// TwinCAT 3 PLC project Untitled1
// ProgramVersion: 3.1.4023.0
// libraries:
//   Tc2_MC2, * (Beckhoff Automation GmbH)
//   Tc2_Standard, * (Beckhoff Automation GmbH)
//   Tc2_System, * (Beckhoff Automation GmbH)
//   Tc2_Utilities, * (Beckhoff Automation GmbH)
//   Tc3_JsonXml, * (Beckhoff Automation GmbH)
//   Tc3_Module, * (Beckhoff Automation GmbH)
// project tree:
//   DUTs/ Bundle.TcDUT, Interval.TcDUT (not stored), PositionMaterials.TcDUT, SuctionPad.TcDUT
//   DUTs/Enums/ A22.TcDUT (not stored), Cardboard.TcDUT (not stored), CornerGuard.TcDUT (not stored), Homing.TcDUT (not stored), SectionEnum.TcDUT, Surface.TcDUT
//   DUTs/Insertion/ABSTRACT/ FBA_Drive.TcPOU, I_ContinuousDrive.TcIO (not stored), I_Drive.TcIO, I_EncodedDrive.TcIO (not stored), I_PositionalDrive.TcIO (not stored)
//   DUTs/Insertion/Drives/ ClearLinkMC.TcPOU, ServoNC.TcPOU, SimplePiston.TcPOU (not stored)
//   DUTs/Insertion/ Insertion.TcPOU
//   DUTs/Machines/ FoldingMachine.TcPOU, KukaRobot.TcPOU (not stored), RobotA22.TcPOU (not stored), WrapMachine.TcPOU (not stored)
//   DUTs/Material Holders/ MaterialHolder.TcPOU (not stored), MaterialSlot.TcDUT, SkidMagazine.TcPOU (not stored)
//   GVLs/ ContainerArrays.TcGVL, GVL.TcGVL (not stored), Hardware.TcGVL, Misc.TcGVL (not stored)
//   / PlcTask.TcTTO
//   POUs/A22 - Cardboard-Corner Guard/AOIs/ AOI_LoadCornerCardboard.TcPOU, AOI_LoadCornerGuard.TcPOU, AOI_LoadFlatCardboard.TcPOU
//   POUs/A22 - Cardboard-Corner Guard/ FiberboardEx.TcPOU
//   POUs/ FB_System.TcPOU, MAIN.TcPOU, BundleToJson.TcPOU
//   POUs/Hardware Calls/ SuctionQualityPtrArr.TcPOU (not stored), SetSuctionsPtrArr.TcPOU (not stored), CallHardwareModules.TcPOU, SuctionQuality.TcPOU (not stored), SetSuctions.TcPOU, SetupHardware.TcPOU (not stored)
//   POUs/Materials/ GetMaterialLength.TcPOU, GetMaterialLengthFromCode.TcPOU (not stored), GetPairMasterLength.TcPOU (not stored), GetPositionMasterLength.TcPOU (not stored), MatchesMaterialType.TcPOU
//   POUs/Utility/ CEILING.TcPOU (not stored), IntegerBitAccess.TcPOU (not stored), IntegerToBoolArray.TcPOU (not stored), WithinTolerance.TcPOU (not stored)
// real-time tasks:
//   TASK PlcTask: cycle T#10ms, priority 20, ADS port 350
// motion (NC):
//   TASK NC-Task 1 SAF: cycle T#2ms, priority 4, ADS port 501
//   TASK NC-Task 1 SVB: cycle T#10ms, priority 8, ADS port 511
//   AXIS A22_IM_HS_L (id 1)
//     OtherSettings: AllowMotionCmdToSlave=true
//     encoder EncType=1
//     drive DrvType=5
//       Analog: TorqueSetpointScale=10, ScaleFactorActTorque=0.1
//       TimeComp: TaskDelayCycles=1
//     controller CtrType=1
//       CtrPara: PriorControlFactor=1
//         Observer: BandWidth=20
//   AXIS A22_IM_HS_R (id 2)
//     OtherSettings: AllowMotionCmdToSlave=true
//     encoder EncType=19
//       EncPara: MaxCount=#xffffffff
//     drive DrvType=16
//       DrvPara: MaxCount=#xffffffff, DriveControlDWord=#x00000100
//         Analog: TorqueSetpointScale=10, ScaleFactorActTorque=0.1
//         TimeComp: TaskDelayCycles=1
//     controller CtrType=1
//       CtrPara: PriorControlFactor=1
//         Observer: BandWidth=20
// I/O:
//   DEVICE Device 2 (TC3 EIP Scanner), AmsNetId 5.131.216.41.4.1
//     ClearLink_A22 // <INFO> 169.254.0.152, ClearLink (ProdCode: 1, Rev: 2.93, Mac: 24:15:10:b0:30:37) </INFO> <EDS> C:\TwinCAT\3.1\Config\Io\EtherNetIP\clearlink_2.92.eds </EDS>
//   DEVICE Device 1 (EtherCAT), AmsNetId 5.131.216.41.2.1
//     EK1200 [EK1200-5000 EtherCAT Power supply (2A E-Bus)]
//       IPC_O [EL2809 16Ch. Dig. Output 24V, 0.5A]
//       JUNC_1 [EK1122 2 port EtherCAT junction]
//         A21_C4 [EK1100 EtherCAT Coupler (2A E-Bus)]
//           A21_C4_I1 [EL1809 16Ch. Dig. Input 24V, 3ms]
//           A21_C4_O2 [EL2809 16Ch. Dig. Output 24V, 0.5A]
//           A21_C4_O3 [EL2809 16Ch. Dig. Output 24V, 0.5A]
//           BRIDGE_ROBOT1 [EL6695 EtherCAT Bridge terminal (Primary)]
//           A21_C4_END [EL9011 End Terminal]
//         A21_SB01 [EP1809-0021 16 Ch. Dig. Input 24V, 3ms, M8]
//         A21_SB05 [EP1008-0001 8 Ch. Dig. Input 24V, 3ms, M8]
//         A21_SB04 [EP1809-0021 16 Ch. Dig. Input 24V, 3ms, M8]
//         A21_SB03 [EP1008-0001 8 Ch. Dig. Input 24V, 3ms, M8]
//         A21_C1 [EK1100 EtherCAT Coupler (2A E-Bus)]
//           A21_C1_I1 [EL1809 16Ch. Dig. Input 24V, 3ms]
//           A21_C1_O2 [EL2809 16Ch. Dig. Output 24V, 0.5A]
//           BRIDGE_ROBOT2 [EL6695 EtherCAT Bridge terminal (Primary)]
//           A21_C1_END [EL9011 End Terminal]
//         A21_SB02 [EP1809-0021 16 Ch. Dig. Input 24V, 3ms, M8]
//         A21_SB07 [EP1008-0001 8 Ch. Dig. Input 24V, 3ms, M8]
//         A21_SB06 [EP1008-0001 8 Ch. Dig. Input 24V, 3ms, M8]
//       JUNC_2 [EK1122 2 port EtherCAT junction]
//         A22_C1 [EK1100 EtherCAT Coupler (2A E-Bus)]
//           A22_C1_I1 [EL1809 16Ch. Dig. Input 24V, 3ms]
//           A22_C1_O2 [EL2809 16Ch. Dig. Output 24V, 0.5A]
//           A22_C1_JUNC [EK1122 2 port EtherCAT junction]
//             A22_C4 [EK1100 EtherCAT Coupler (2A E-Bus)]
//               A22_C4_I1 [EL1809 16Ch. Dig. Input 24V, 3ms]
//               A22_C4_O2 [EL2809 16Ch. Dig. Output 24V, 0.5A]
//               A22_C4_O3 [EL2809 16Ch. Dig. Output 24V, 0.5A]
//               Term 31 (EL9011) [EL9011 End Terminal]
//             A22_C4_NC2 [CD02 EtherCAT Drive (CoE)]
//             A22_C4_NC1_TEMP [EK1100 EtherCAT Coupler (2A E-Bus)]
//               Term 34 (EL1008) [EL1008 8Ch. Dig. Input 24V, 3ms]
//               Term 35 (EL2008) [EL2008 8Ch. Dig. Output 24V, 0.5A]
//               Term 36 (EL9011) [EL9011 End Terminal]
//             A22_SB01 [EP1809-0021 16 Ch. Dig. Input 24V, 3ms, M8]
//             A22_SB04 [EP1809-0021 16 Ch. Dig. Input 24V, 3ms, M8]
//             A22_SB05 [EP1008-0001 8 Ch. Dig. Input 24V, 3ms, M8]
//             A22_C5 [EK1100 EtherCAT Coupler (2A E-Bus)]
//               A22_C5_I1 [EL1809 16Ch. Dig. Input 24V, 3ms]
//               A22_C5_O2 [EL2809 16Ch. Dig. Output 24V, 0.5A]
//               A22_C5_END [EL9011 End Terminal]
//             A22_SB06 [EP1008-0001 8 Ch. Dig. Input 24V, 3ms, M8]
//             A22_C6 [EK1100 EtherCAT Coupler (2A E-Bus)]
//               A22_C6_I1 [EL1809 16Ch. Dig. Input 24V, 3ms]
//               A22_C6_O2 [EL2809 16Ch. Dig. Output 24V, 0.5A]
//               A22_C6_O3 [EL2809 16Ch. Dig. Output 24V, 0.5A]
//               BRDIGE_ROBOT3 [EL6695 EtherCAT Bridge terminal (Primary)]
//               A22_C6_END [EL9011 End Terminal]
//             A22_SB08 [EP1008-0001 8 Ch. Dig. Input 24V, 3ms, M8]
//             A22_SB09 [EP2338-1001 8 Ch. Dig. Input/Output 24V, 3ms, 0,5A, M8]
//             A22_SB03 [EP1008-0001 8 Ch. Dig. Input 24V, 3ms, M8]
//             A22_SB02 [EP1809-0021 16 Ch. Dig. Input 24V, 3ms, M8]
//             A22_SB07 [EP1008-0001 8 Ch. Dig. Input 24V, 3ms, M8]
//             A22_C7 [EK1100 EtherCAT Coupler (2A E-Bus)]
//               A22_C7_I1 [EL1809 16Ch. Dig. Input 24V, 3ms]
//               A22_C7_O2 [EL2809 16Ch. Dig. Output 24V, 0.5A]
//               BRIDGE_ROBOT4 [EL6695 EtherCAT Bridge terminal (Primary)]
//               A22_C7_END [EL9011 End Terminal]
// variable links:
//   NC-Task 1 SAF/Axes/A22_IM_HS_R <-> Device 1 (EtherCAT)/EK1200/JUNC_2/A22_C1/A22_C1_JUNC/A22_C4_NC2
//     Drive/Inputs/In/nDataIn1 <-> TxPDO 1/Following Error Actual Value
//     Drive/Inputs/In/nDataIn3[0] <-> TxPDO 4/Torque Actual Value
//     Drive/Inputs/In/nDcOutputTime <-> InfoData/DcOutputShift
//     Drive/Inputs/In/nState1 <-> TxPDO 4/Statusword
//     Drive/Inputs/In/nState2 <-> TxPDO 4/Statusword @bit 8
//     Drive/Inputs/In/nState4 @bit 1 <-> WcState/InputToggle
//     Drive/Inputs/In/nState4 <-> WcState/WcState
//     Drive/Inputs/In/nState5 <-> TxPDO 3/Modes of Operation Display
//     Drive/Outputs/Out/nCtrl1 <-> RxPDO 4/Controlword
//     Drive/Outputs/Out/nCtrl2 <-> RxPDO 4/Controlword @bit 8
//     Drive/Outputs/Out/nCtrl5 <-> RxPDO 4/Modes of Operation
//     Drive/Outputs/Out/nDataOut1 <-> RxPDO 1/Target Position
//     Drive/Outputs/Out/nDataOut2 <-> RxPDO 2/Target Velocity
//     Drive/Outputs/Out/nDataOut3[0] <-> RxPDO 4/Torque Offset
//     Drive/Outputs/Out/nDataOut4[0] <-> RxPDO 3/Target Torque
//     Enc/Inputs/In/nDataIn1 <-> TxPDO 2/Position Actual Value
//     Enc/Inputs/In/nDcInputTime <-> InfoData/DcInputShift
//     Enc/Inputs/In/nState4 @bit 1 <-> WcState/InputToggle
//     Enc/Inputs/In/nState4 <-> WcState/WcState
//   Untitled1/Untitled1 Instance <-> Device 1 (EtherCAT)/EK1200/JUNC_2/A22_C1/A22_C1_JUNC/A22_C4/A22_C4_O3
//     PlcTask Outputs/Hardware.verticalDriveA22Right.brakeRelease <-> Channel 1/Output
//   Untitled1/Untitled1 Instance <-> Device 1 (EtherCAT)/EK1200/JUNC_2/A22_C1/A22_C1_JUNC/A22_C6/BRDIGE_ROBOT3
//     PlcTask Inputs/Hardware.robot3.inputs[{2..20}] <-> IO Inputs/In_{2..20}  (19 links)
//     PlcTask Inputs/Hardware.robot3.inputs[1] <-> IO Inputs/In
//     PlcTask Inputs/Hardware.robot3.offline <-> SYNC Inputs/External device not connected
//     PlcTask Outputs/Hardware.robot3.outputs[{2..20}] <-> IO Outputs/Out_{2..20}  (19 links)
//     PlcTask Outputs/Hardware.robot3.outputs[1] <-> IO Outputs/Out
//   Untitled1/Untitled1 Instance <-> Device 1 (EtherCAT)/EK1200/JUNC_2/A22_C1/A22_C1_JUNC/A22_C7/BRIDGE_ROBOT4
//     PlcTask Inputs/Hardware.robot4.inputs[{2..20}] <-> IO Inputs/In_{2..20}  (19 links)
//     PlcTask Inputs/Hardware.robot4.inputs[1] <-> IO Inputs/In
//     PlcTask Inputs/Hardware.robot4.offline <-> SYNC Inputs/External device not connected
//     PlcTask Outputs/Hardware.robot4.outputs[{2..20}] <-> IO Outputs/Out_{2..20}  (19 links)
//     PlcTask Outputs/Hardware.robot4.outputs[1] <-> IO Outputs/Out
//   Untitled1/Untitled1 Instance <-> Device 1 (EtherCAT)/EK1200/JUNC_2/A22_C1/A22_C1_JUNC/A22_SB01
//     PlcTask Inputs/Hardware.horizontalDriveA22Left.home <-> Channel 6/Input
//     PlcTask Inputs/Hardware.horizontalDriveA22Left.innerLimit <-> Channel 5/Input
//     PlcTask Inputs/Hardware.horizontalDriveA22Left.outerLimit <-> Channel 4/Input
//     PlcTask Inputs/Hardware.suctionA22BottomLeft[1].occupied <-> Channel 10/Input
//     PlcTask Inputs/Hardware.suctionA22BottomLeft[2].occupied <-> Channel 11/Input
//     PlcTask Inputs/Hardware.suctionA22BottomLeft[3].occupied <-> Channel 12/Input
//     PlcTask Inputs/Hardware.suctionA22TopLeft[1].occupied <-> Channel 7/Input
//     PlcTask Inputs/Hardware.suctionA22TopLeft[2].occupied <-> Channel 8/Input
//     PlcTask Inputs/Hardware.suctionA22TopLeft[3].occupied <-> Channel 9/Input
//     PlcTask Inputs/Hardware.verticalDriveA22Left.home <-> Channel 3/Input
//     PlcTask Inputs/Hardware.verticalDriveA22Left.innerLimit <-> Channel 2/Input
//     PlcTask Inputs/Hardware.verticalDriveA22Left.outerLimit <-> Channel 1/Input
//   Untitled1/Untitled1 Instance <-> Device 1 (EtherCAT)/EK1200/JUNC_2/A22_C1/A22_C1_JUNC/A22_SB02
//     PlcTask Inputs/Hardware.horizontalDriveA22Right.home <-> Channel 6/Input
//     PlcTask Inputs/Hardware.horizontalDriveA22Right.innerLimit <-> Channel 4/Input
//     PlcTask Inputs/Hardware.horizontalDriveA22Right.outerLimit <-> Channel 5/Input
//     PlcTask Inputs/Hardware.suctionA22BottomRight[1].occupied <-> Channel 10/Input
//     PlcTask Inputs/Hardware.suctionA22BottomRight[2].occupied <-> Channel 11/Input
//     PlcTask Inputs/Hardware.suctionA22BottomRight[3].occupied <-> Channel 12/Input
//     PlcTask Inputs/Hardware.suctionA22TopRight[1].occupied <-> Channel 7/Input
//     PlcTask Inputs/Hardware.suctionA22TopRight[2].occupied <-> Channel 8/Input
//     PlcTask Inputs/Hardware.suctionA22TopRight[3].occupied <-> Channel 9/Input
//     PlcTask Inputs/Hardware.verticalDriveA22Right.home <-> Channel 3/Input
//     PlcTask Inputs/Hardware.verticalDriveA22Right.innerLimit <-> Channel 2/Input
//     PlcTask Inputs/Hardware.verticalDriveA22Right.outerLimit <-> Channel 1/Input
//   Untitled1/Untitled1 Instance <-> Device 1 (EtherCAT)/EK1200/JUNC_2/A22_C1/A22_C1_JUNC/A22_SB06
//     PlcTask Inputs/Hardware.magazineA22Left.inPosition[1] <-> Channel 7/Input
//     PlcTask Inputs/Hardware.magazineA22Left.inPosition[2] <-> Channel 8/Input
//   Untitled1/Untitled1 Instance <-> Device 2 (TC3 EIP Scanner)/ClearLink_A22
//     PlcTask Inputs/Hardware.verticalDriveA22Left.hlfb <-> Connection 1 (Input/Output)/Inputs/Motor0 HLFB Duty
//     PlcTask Inputs/Hardware.verticalDriveA22Right.hlfb <-> Connection 1 (Input/Output)/Inputs/Motor1 HLFB Duty
//     PlcTask Outputs/Hardware.verticalDriveA22Left.outputRegister <-> Connection 1 (Input/Output)/Outputs/Motor0 Out Reg
//     PlcTask Outputs/Hardware.verticalDriveA22Left.pulse <-> Connection 1 (Input/Output)/Outputs/Motor0 Trig Pulses
//     PlcTask Outputs/Hardware.verticalDriveA22Right.outputRegister <-> Connection 1 (Input/Output)/Outputs/Motor1 Out Reg
//     PlcTask Outputs/Hardware.verticalDriveA22Right.pulse <-> Connection 1 (Input/Output)/Outputs/Motor1 Trig Pulses
//   Untitled1/Untitled1 Instance <-> NC-Task 1 SAF/Axes/A22_IM_HS_L
//     PlcTask Inputs/Hardware.horizontalDriveA22Left.axis.NcToPlc <-> Outputs/ToPlc
//     PlcTask Outputs/Hardware.horizontalDriveA22Left.axis.PlcToNc <-> Inputs/FromPlc
//   Untitled1/Untitled1 Instance <-> NC-Task 1 SAF/Axes/A22_IM_HS_R
//     PlcTask Inputs/Hardware.horizontalDriveA22Right.axis.NcToPlc <-> Outputs/ToPlc
//     PlcTask Outputs/Hardware.horizontalDriveA22Right.axis.PlcToNc <-> Inputs/FromPlc

CONFIGURATION Untitled1
    RESOURCE PLC ON TwinCAT3
        TASK PlcTask(INTERVAL := T#10ms, PRIORITY := 20);
        PROGRAM MAIN WITH PlcTask : MAIN;
    END_RESOURCE
END_CONFIGURATION

// ---- DUTs/Bundle.TcDUT
{attribute 'enable_dynamic_creation'}
TYPE Bundle :
STRUCT
	id : STRING;
	weight : REAL;
	
	length : INT;
	width : INT;
	height : INT;
	
	pieces : INT;
	layers : INT;
	piecesPerLayer : INT;
	
	extrusionWeight : INT;
	extrusionHeight : INT;
	extrusionWidth : INT;
	
	//if a process is true, send it to the correct area and turn it false when complete
	reqProcesses : ARRAY[0..3] OF BOOL; //this may not be used
	
	manRE, autoRE : BOOL; //repacking - coming soon
	manSS, autoSS : BOOL; //packaging
	
	paperFront : BOOL;
	paperBack : BOOL;
	cardboardFront : BOOL;
	cardboardBack : BOOL;
	
	paperTop : ARRAY[0..GVL.maxPairs] OF Interval;
	paperLeft : ARRAY[0..GVL.maxPairs] OF Interval;
	paperRight : ARRAY[0..GVL.maxPairs] OF Interval;
	paperBottom : ARRAY[0..GVL.maxPairs] OF Interval;
		
	cardboard : ARRAY[0..GVL.maxPairs] OF PositionMaterials;
	cardboardTopLeftFold : ARRAY[0..GVL.maxPairs] OF INT;
	cardboardTopRightFold : ARRAY[0..GVL.maxPairs] OF INT;
	cardboardBottomLeftFold : ARRAY[0..GVL.maxPairs] OF INT;
	cardboardBottomRightFold : ARRAY[0..GVL.maxPairs] OF INT;
	
	topLeftFolds : ARRAY[0..GVL.maxPairs] OF INT;
	topRightFolds : ARRAY[0..GVL.maxPairs] OF INT;
	bottomLeftFolds : ARRAY[0..GVL.maxPairs] OF INT;
	bottomRightFolds : ARRAY[0..GVL.maxPairs] OF INT;
	
	cornerGuard : ARRAY[0..GVL.maxPairs] OF PositionMaterials;
	
	chipboard : ARRAY[0..GVL.maxPairs] OF PositionMaterials;
	woodBunk : ARRAY[0..GVL.maxPairs] OF PositionMaterials;
	
	cardboard_over_cornerGuard : BOOL;
	
	currStep : USINT; //for runtime use only
	
	//for production log database
	
	timeStart : TIMESTRUCT;
	timeDone : TIMESTRUCT;
END_STRUCT
END_TYPE

// ---- DUTs/Enums/SectionEnum.TcDUT
{attribute 'qualified_only'}
TYPE SectionEnum :
(
	NULL_SECTION := 0,
	PAPER,
	CARDBOARD_CORNERGUARD,
	CHIPBOARD,
	WOOD_BUNK,
	OUTPUT,
	
	size
);
END_TYPE

// ---- DUTs/Enums/Surface.TcDUT
{attribute 'qualified_only'}
//{attribute 'strict'}
TYPE Surface :
(
	NULL,
	
	TOP,
	LEFT,
	RIGHT,
	BOTTOM,
	
	TOP_LEFT,
	TOP_RIGHT,
	BOTTOM_LEFT,
	BOTTOM_RIGHT,
	
	size
);
END_TYPE

// ---- DUTs/Material Holders/MaterialSlot.TcDUT
TYPE MaterialSlot :
STRUCT
	material : STRING;
	occupied AT %I* : BOOL;
END_STRUCT
END_TYPE

// ---- DUTs/PositionMaterials.TcDUT
TYPE PositionMaterials :
STRUCT
	position : REAL; //:= GVL.nullPos; //default value is set to predefined constant if bundle needs less than 16+1 position material pairs
	
	top : STRING;
	right : STRING;
	left : STRING;
	//sides : STRING;
	bottom : STRING;
	
	topLeft : STRING;
	topLeftFold : USINT;
	
	topRight : STRING;
	topRightFold : USINT;
	
	bottomLeft : STRING;
	bottomLeftFold : USINT;
	
	bottomRight : STRING;
	bottomRightFold : USINT;

	wrapPoints : USINT;
	wrapRotations : USINT;
END_STRUCT
END_TYPE

// ---- DUTs/SuctionPad.TcDUT
TYPE SuctionPad :
STRUCT
	enable AT %Q* : BOOL;
	occupied AT %I* : BOOL;
END_STRUCT
END_TYPE

// ---- GVLs/ContainerArrays.TcGVL
//{attribute 'qualified_only'}
VAR_GLOBAL //data arrays to be passed into material holder FBs - do not access directly
	skidHmiA22Left : ARRAY[1...Cardboard.size-1] OF MaterialSlot;
	skidHmiA22Right : ARRAY[1...Cardboard.size-1] OF MaterialSlot;
	
	magazineHmiA22Left : ARRAY[1..CornerGuard.size-1] OF MaterialSlot;
	magazineHmiA22Right : ARRAY[1..CornerGuard.size-1] OF MaterialSlot;
END_VAR

// ---- GVLs/Hardware.TcGVL
//{attribute 'qualified_only'}
VAR_GLOBAL //complete modules
	robot3, robot4 : RobotA22;
	
	benderA22Left : FoldingMachine;
	
	skidA22Left, skidA22Right : SkidMagazine;
	magazineA22Left, magazineA22Right : SkidMagazine;
	
	wrapperA22 : WrapMachine;
	
	horizontalDriveA22Left, horizontalDriveA22Right : ServoNC := (
		limitSensorDefaultState := TRUE);
		
	verticalDriveA22Left, verticalDriveA22Right : ClearLinkMC := (
		limitSensorDefaultState := TRUE, 
		homingDirection := TRUE, //outwards (up)
		minPosition := 0,
		displacementPerRotation := 1,
		unitsPerPulse := 800); //800 counts = 1 rotation
		
	insertionA22Left, insertionA22Right : Insertion;
		
	pistonA22Bottom : SimplePiston;
	
	(*
	each of these suction arrays are composed of 3 pads
	pad [2] is the corner pad used for corner guards
	pads [1] and [3] are the outer pads used for corner cardboards
	*)
	suctionA22TopLeft : ARRAY[1..3] OF SuctionPad;
	suctionA22TopRight : ARRAY[1..3] OF SuctionPad;
	suctionA22BottomLeft : ARRAY[1..3] OF SuctionPad; 
	suctionA22BottomRight : ARRAY[1..3] OF SuctionPad;
	
	suctionA22Bottom : ARRAY[1..2] OF SuctionPad;
END_VAR

// ---- DUTs/Insertion/ABSTRACT/I_Drive.TcIO
INTERFACE I_Drive

{attribute 'monitoring':='call'}
PROPERTY ABSTRACT Active : BOOL
GET
END_GET
END_PROPERTY

{attribute 'monitoring':='call'}
PROPERTY ABSTRACT AtHome : BOOL
GET
END_GET
END_PROPERTY

{attribute 'monitoring':='call'}
PROPERTY ABSTRACT AtInnerLimit : BOOL
GET
END_GET
END_PROPERTY

{attribute 'monitoring':='call'}
PROPERTY ABSTRACT AtOuterLimit : BOOL
GET
END_GET
END_PROPERTY

{attribute 'monitoring':='call'}
PROPERTY ABSTRACT Contact : BOOL
GET
END_GET
END_PROPERTY

{attribute 'monitoring':='call'}
PROPERTY ABSTRACT Error : BOOL
GET
END_GET
END_PROPERTY

{attribute 'monitoring':='call'}
PROPERTY ABSTRACT HomeSet : BOOL
GET
END_GET
END_PROPERTY

METHOD ABSTRACT homingSequence : BOOL
VAR_INPUT
END_VAR
END_METHOD

METHOD ABSTRACT stop : BOOL
VAR_INPUT
END_VAR
END_METHOD

END_INTERFACE

// ---- POUs/MAIN.TcPOU
PROGRAM MAIN
VAR_OUTPUT
	currentTime : TIMESTRUCT;
END_VAR
VAR
	execute : BOOL;
	manualStep : BOOL := TRUE;
	manualSuction : BOOL := FALSE;
	stop : BOOL;
	
	moduleA22 : FiberboardEx;
END_VAR
VAR
	getLocalTime : FB_LocalSystemTime;
	test : BOOL;
END_VAR

CallHardwareModules(); //start program with hardware call

SetupHardware(); //setup hardware

callModules(); //call section modules

CallHardwareModules(); //end program with hardware call


//unrelated tests
//BundleToJson();

ACTION callModules:
getLocalTime(
	sNetID:= , 
	bEnable:= TRUE, 
	dwCycle:= , 
	dwOpt:= , 
	tTimeout:= , 
	bValid=> , 
	systemTime=> currentTime, 
	tzID=> );

moduleA22(
	execute:= execute, 
	stop:= stop, 
	manualStep:= manualStep, 
	manualSuction:= manualSuction, 
	
	benderLeft:= benderA22Left, 
	robotLeft:= robot3, 
	robotRight:= robot4, 
	skidLeft:= skidA22Left, 
	skidRight:= skidA22Right, 
	magazineLeft:= magazineA22Left, 
	magazineRight:= magazineA22Right, 
	wrapper:= wrapperA22,
	insertionLeft:= insertionA22Left, 
	insertionRight:= insertionA22Right,
	pistonBottom:= pistonA22Bottom, 
	suctionTopLeft:= suctionA22TopLeft, 
	suctionTopRight:= suctionA22TopRight, 
	suctionBottomLeft:= suctionA22BottomLeft, 
	suctionBottomRight:= suctionA22BottomRight, 
	suctionBottom:= suctionA22Bottom,
	
	generalError=> , 
	failLeft=> , 
	failRight=> );
END_ACTION

END_PROGRAM

// ---- POUs/A22 - Cardboard-Corner Guard/FiberboardEx.TcPOU
FUNCTION_BLOCK FiberboardEx
VAR_IN_OUT //controls
	execute : BOOL;
	stop : BOOL;
	
	manualStep : BOOL;
	manualSuction : BOOL;
END_VAR
VAR_IN_OUT
	benderLeft : FoldingMachine;
	
	robotLeft, robotRight : RobotA22;
	
	skidLeft, skidRight : SkidMagazine;
	magazineLeft, magazineRight : SkidMagazine;
	
	wrapper : WrapMachine;
	
	insertionLeft, insertionRight : Insertion;
	pistonBottom : SimplePiston;
	
	suctionTopLeft : ARRAY[*] OF SuctionPad; (*1..3*)
	suctionTopRight : ARRAY[*] OF SuctionPad; (*1..3*)
	suctionBottomLeft : ARRAY[*] OF SuctionPad; (*1..3*)
	suctionBottomRight : ARRAY[*] OF SuctionPad; (*1..3*)
	
	suctionBottom : ARRAY[*] OF SuctionPad; (*1..2*)
END_VAR
VAR_OUTPUT
	generalError : BOOL;
	failLeft, failRight : BOOL;
END_VAR
VAR //for testing only
	latchLeft, latchRight : BOOL; //prevents sliders from overshooting the inner limit sensor
	
	suctionEnableTopLeft : BOOL;
	suctionEnableTopRight : BOOL;
	suctionEnableBottomLeft : BOOL;
	suctionEnableBottomRight : BOOL;
	
	ready : BOOL;
	done : BOOL;
END_VAR
VAR	
	step : (IDLE, LOAD_CORNERS, LOAD_FLATS, PUSH, TARGET_WRAP_POSITION, WRAP_AND_RELEASE, COMPLETE := 1050);
	iPair : INT;
	
	masterLoadStep : INT;
	loadStepLeft, loadStepRight : INT;
	
	iWrap : INT;
	wrapPoints : INT;
	wrapRotations : INT;
	masterLength : INT;
	
	releaseDelayTimer : TON;
END_VAR
VAR //local types
	topLeftFoldsArr, topRightFoldsArr, bottomLeftFoldsArr, bottomRightFoldsArr : ARRAY[0..GVL.maxPairs] OF INT;
	materialsArr : ARRAY[0..GVL.maxPairs] OF PositionMaterials := [
		(
			position := 0,
			top := 'CAR20M',
			left := 'CAR20S',
			right := 'CAR20S',
			bottom := 'CAR20L',
			topLeft := 'CAR28M',
			topRight := 'CAR28S',
			bottomLeft := 'CAR28S',
			bottomRight := 'CAR28L',
			wrapPoints := 1,
			wrapRotations := 4
		),
		(
			position := 0,
			topLeft := 'COR48',
			topRight := 'COR48',
			bottomLeft := 'COR48',
			bottomRight := 'COR48'
		)];
	
	demoHeight : REAL := 600; //600mm, 60cm
	
	innerLoadedMaterials, outerLoadedMaterials : ARRAY[Surface.TOP..Surface.BOTTOM_RIGHT] OF STRING;
	//inner: cardboard by default
	//outer: corner guard by default
END_VAR
VAR CONSTANT
	sectionID : SectionEnum := SectionEnum.CARDBOARD_CORNERGUARD;
	releaseDelay : TIME := T#2000MS;
END_VAR
VAR
	//AOIs encapsulate functionality and reduce the number of module variables
	aoiCornerGuardLeft, aoiCornerGuardRight : AOI_LoadCornerGuard;
	aoiCornerCardboardLeft, aoiCornerCardboardRight : AOI_LoadCornerCardboard;
	aoiFlatCardboardLeft, aoiFlatCardboardRight : AOI_LoadFlatCardboard;
END_VAR

{warning disable C0371}
(*
corrected sequence:
	load sides
	load corners
	load bottom
	load top
*)

CASE step OF
	IDLE:
		IF execute THEN
			execute := FALSE;
			step := LOAD_CORNERS;
		END_IF
	
	LOAD_CORNERS:
		IF
			(auto AND done) OR
			(NOT auto AND execute)
		THEN
			aoiCornerCardboardLeft.reset();
			aoiCornerCardboardRight.reset();
			
			aoiCornerGuardLeft.reset();
			aoiCornerGuardRight.reset();
			
			aoiFlatCardboardLeft.reset();
			aoiFlatCardboardRight.reset();
			
			step := LOAD_FLATS;
			RETURN;
		END_IF
		
		IF NOT done THEN
			done := load(pairIndex := iPair);
		END_IF
		
	LOAD_FLATS:
		IF
			(auto AND done) OR
			(NOT auto AND execute)
		THEN
			aoiCornerCardboardLeft.reset();
			aoiCornerCardboardRight.reset();
			
			aoiCornerGuardLeft.reset();
			aoiCornerGuardRight.reset();
			
			aoiFlatCardboardLeft.reset();
			aoiFlatCardboardRight.reset();
			
			step := PUSH;
			RETURN;
		END_IF
		
		IF NOT done THEN
			done := loadFlatCardboards(pairIndex := iPair);
		END_IF
		
	PUSH:
		IF
			(auto AND latchLeft AND latchRight AND pistonBottom.extended) OR
			(insertionLeft.contact AND insertionRight.contact AND pistonBottom.extended) OR
			(NOT auto AND execute)
		THEN
			step := TARGET_WRAP_POSITION;
			RETURN;
		END_IF
		
		IF //align slider to 5mm gap above bundle height
			NOT insertionLeft.align(1000-demoHeight+5) OR
			NOT insertionRight.align(1000-demoHeight+5)
		THEN
			RETURN;
		END_IF
		
		insertionLeft.press();
		insertionRight.press();
		pistonBottom.extend();
		
	TARGET_WRAP_POSITION:		
		IF iWrap >= wrapPoints THEN
			step := COMPLETE;
			RETURN;
		END_IF
		
		//loadNextPair := materialsArr[iPair].position = materialsArr[iPair + 1].position;	
		
		IF materialsArr[iPair].position = materialsArr[iPair + 1].position THEN
			masterLength := MAX( GetPairMasterLength(materialsArr[iPair]), GetPairMasterLength(materialsArr[iPair + 1]) );
			wrapPoints := MAX( materialsArr[iPair].wrapPoints, materialsArr[iPair + 1].wrapPoints );
			wrapRotations := MAX( materialsArr[iPair].wrapRotations, materialsArr[iPair + 1].wrapRotations );
		ELSE
			masterLength := GetPairMasterLength(materialsArr[iPair]);
			wrapPoints := materialsArr[iPair].wrapPoints;
			wrapRotations := materialsArr[iPair].wrapRotations;
		END_IF
		
		(*
		directionCheckAndSet(
			wrapConveyorPos,
			(currentPair.position - masterLength/2) + (masterLength/(currentPair.wrapPoints + 1) * (iWrap + 1)));
		*)
		step := WRAP_AND_RELEASE;
		
	WRAP_AND_RELEASE:
		releaseDelayTimer(IN:= , PT:= releaseDelay, Q=> , ET=> );
		
		IF wrapper.ready THEN
			wrapper.wrap(wrapRotations);
			releaseDelayTimer.IN := TRUE;
		END_IF
		
		IF releaseDelayTimer.Q THEN
			SetSuctions(suctions := suctionTopLeft, state := FALSE);
			SetSuctions(suctions := suctionTopRight, state := FALSE);
			SetSuctions(suctions := suctionBottomLeft, state := FALSE);
			SetSuctions(suctions := suctionBottomRight, state := FALSE);
			
			insertionLeft.align(0);
			insertionRight.align(0);
			insertionLeft.release();
			insertionRight.release();
			
			pistonBottom.retract();
		END_IF
		
		IF wrapper.done AND insertionLeft.home AND insertionRight.home AND pistonBottom.retracted THEN
			releaseDelayTimer.IN := FALSE;
			step := WRAP_AND_RELEASE;
		END_IF
	
	COMPLETE:
		iPair := (iPair + 1) MOD GVL.maxPairs;
		iWrap := wrapPoints := wrapRotations := 0;
		step := IDLE;
		
END_CASE

ACTION blocks:
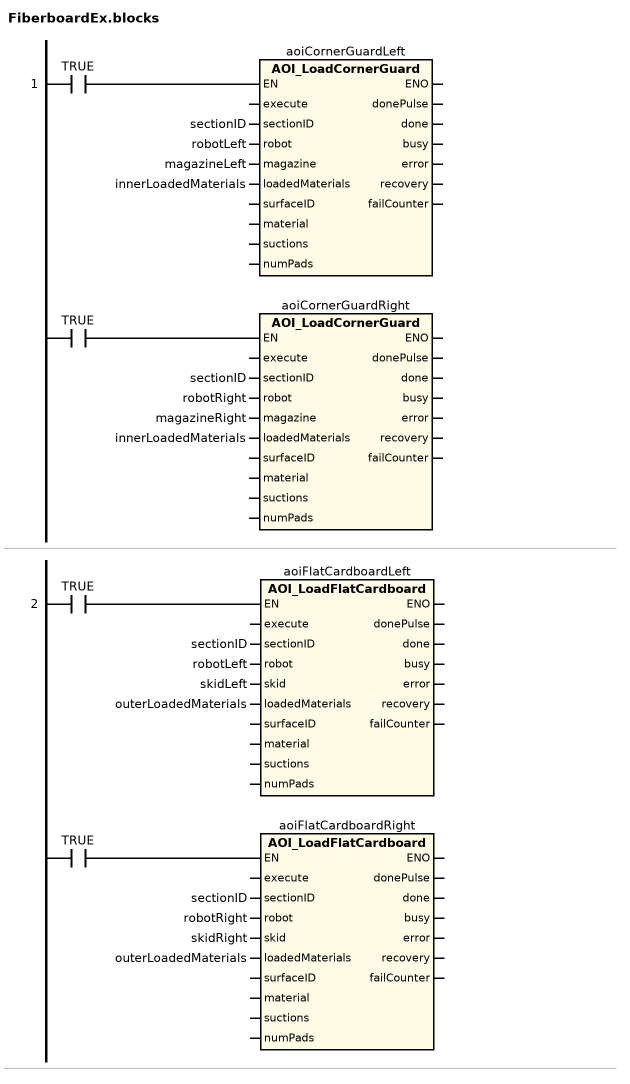
// NETWORK 1
aoiCornerGuardLeft(
    sectionID := sectionID,
    robot := robotLeft,
    magazine := magazineLeft,
    loadedMaterials := innerLoadedMaterials); // AOI_LoadCornerGuard
aoiCornerGuardRight(
    sectionID := sectionID,
    robot := robotRight,
    magazine := magazineRight,
    loadedMaterials := innerLoadedMaterials); // AOI_LoadCornerGuard

// NETWORK 2
aoiFlatCardboardLeft(
    sectionID := sectionID,
    robot := robotLeft,
    skid := skidLeft,
    loadedMaterials := outerLoadedMaterials); // AOI_LoadFlatCardboard
aoiFlatCardboardRight(
    sectionID := sectionID,
    robot := robotRight,
    skid := skidRight,
    loadedMaterials := outerLoadedMaterials); // AOI_LoadFlatCardboard
END_ACTION

ACTION callLocalModules:
{warning disable C0371}
END_ACTION

ACTION homingSequence:
insertionLeft.homingSequence();
insertionRight.homingSequence();
pistonBottom.retract();
END_ACTION

METHOD PROTECTED leftCornerSequence : BOOL
VAR_IN_OUT
	robot : RobotA22;
	skid : SkidMagazine;
	suctions : POINTER TO SuctionPad; //ARRAY[*] OF SuctionPad;
	loadStep : INT;
END_VAR
VAR_INPUT
	surfaceID : Surface;
	material : STRING;
	foldPos0 : INT;
	foldPos1 : INT;
END_VAR
VAR_OUTPUT
	error : BOOL;
END_VAR
VAR
	column : INT;
END_VAR
VAR CONSTANT
	suctionDistance : INT := 10;
END_VAR
(*
{warning disable C0371}
IF material = '' THEN
	leftCornerSequence := TRUE;
	RETURN;
END_IF

benderLeft.setFoldingPositions(foldPos0, foldPos1);

CASE loadStep OF
	0:
		robot.clearCommand();
		IF robot.Ready AND overhead = '' THEN
			loadStep := 10;
		END_IF
		
	10: //skid to bender
		IF NOT skid.findSlot(material:= material, index=> column) THEN
			error := TRUE;
			RETURN;
		END_IF
		
		(*
		IF robot.eoatDistance < suctionDistance THEN
			robot.HoldMaterial := skid.getSlot(i := column);
		END_IF
		*)
		
		IF robot.Done THEN
			loadStep := 20;
			RETURN;
		END_IF
		
		robot.setGroup(group := 1, value := A22.TRANSFER_TO_BENDER);
		robot.setGroup(group := 2, value := foldPos0);
		robot.setGroup(group := 3, value := foldPos1);
		
	20: //bend
		//IF benderLeft.done THEN
			loadStep := 30;
		//END_IF
		
	30: //bender to overhead or left insertion
		IF wrapper.trayOccupied AND wrapper.Overhead = '' AND robot.HoldMaterial <> '' THEN
			wrapper.Overhead := robot.HoldMaterial;
			robot.HoldMaterial := '';
		END_IF
	
		IF robot.Done THEN
			loadStep := COMPLETE;
			RETURN;
		END_IF
		
		CASE surfaceID OF
			Surface.TOP_RIGHT:		robot.setGroup(group := 1, value := A22.TRANSFER_TO_OVERHEAD);
			Surface.BOTTOM_RIGHT:	robot.setGroup(group := 1, value := A22.TRANSFER_TO_OVERHEAD);
			Surface.TOP_LEFT:		robot.setGroup(group := 1, value := A22.LOAD_BENDER_TO_UPPER_CORNER);
			Surface.BOTTOM_LEFT:	robot.setGroup(group := 1, value := A22.LOAD_BENDER_TO_LOWER_CORNER);
		END_CASE
		robot.setGroup(group := 2, value := 0);
		robot.setGroup(group := 3, value := 0);
	
	COMPLETE:
		CASE surfaceID OF
			Surface.TOP_LEFT:		suctionTopLeft[1].enable := suctionTopLeft[3].enable := TRUE;
			Surface.BOTTOM_LEFT:	suctionBottomLeft[1].enable := suctionBottomLeft[3].enable := TRUE;
		END_CASE
		
		leftCornerSequence := TRUE;
		
END_CASE
*)
END_METHOD

METHOD PROTECTED load : BOOL
VAR_INPUT
	pairIndex : INT;
END_VAR
VAR
	pair : REFERENCE TO PositionMaterials REF= materialsArr[pairIndex];
	nextPair : REFERENCE TO PositionMaterials;
END_VAR
(*
unlike other sections, the load() function for cardboard + corner guard only loads the corners
to load flat cardboards, use the function loadFlats()
*)
{warning disable C0371}

IF robotLeft.error OR robotRight.error THEN
	RETURN;
ELSIF NOT (robotLeft.reserve(sectionID) AND robotRight.reserve(sectionID)) THEN //both robots must be reserved first
	RETURN;
END_IF

IF pairIndex + 1 < GVL.maxPairs THEN
	nextPair REF= materialsArr[pairIndex + 1];
END_IF

CASE masterLoadStep OF
	0: //load this pair's side cardboards
		masterLoadStep := 10;
		IF
			loadFlatCardboardsEx(
				robot:= robotLeft, 
				aoiLoad:= aoiFlatCardboardLeft, 
				loadStep:= loadStepLeft, 
				pairIndex:= pairIndex, 
				includeTop:= FALSE, 
				includeLeft:= TRUE, 
				includeRight:= FALSE, 
				includeBottom:= FALSE, 
				error=> )
			AND
			loadFlatCardboardsEx(
				robot:= robotLeft, 
				aoiLoad:= aoiFlatCardboardLeft, 
				loadStep:= loadStepLeft, 
				pairIndex:= pairIndex, 
				includeTop:= FALSE, 
				includeLeft:= FALSE, 
				includeRight:= TRUE, 
				includeBottom:= FALSE, 
				error=> )
		THEN
			masterLoadStep := 10;
			loadStepLeft := loadStepRight := 0;
		END_IF
		
		
	10: //next pair (which is to be placed over this pair) has the same position as this pair
		IF pairIndex + 1 >= GVL.maxPairs THEN //no next pair - final pair is index 15 (16-1), not 16
			masterLoadStep := 20;
			loadStepLeft := loadStepRight := 0;
			
		ELSIF pair.position < nextPair.position THEN
			masterLoadStep := 20;
			loadStepLeft := loadStepRight := 0;
		(*	
		ELSIF MatchesMaterialType(pair:= nextPair, materialType:= 'CAR') AND_THEN loadCornerCardboards(pairIndex:= pairIndex + 1) THEN
			masterLoadStep := 20;
			loadStepLeft := loadStepRight := 0;
		*)
		ELSIF MatchesMaterialType(pair:= nextPair, materialType:= 'COR') AND_THEN loadCornerGuards(pairIndex:= pairIndex + 1) THEN
			masterLoadStep := 20;
			loadStepLeft := loadStepRight := 0;
			
		END_IF
		
	20: //load current pair
		IF
			MatchesMaterialType(pair:= pair, materialType:= 'CAR') AND_THEN loadCornerCardboards(pairIndex:= iPair) OR_ELSE
			MatchesMaterialType(pair:= pair, materialType:= 'COR') AND_THEN loadCornerGuards(pairIndex:= iPair)
		THEN //is cardboard
			loadStepLeft := loadStepRight := 0;
			masterLoadStep := COMPLETE;
		END_IF
	
	COMPLETE:
		robotLeft.release(sectionID);
		robotRight.release(sectionID);
		
		loadStepLeft := loadStepRight := 0;
		masterLoadStep := 0;
		load := TRUE;
	
END_CASE
END_METHOD

METHOD PROTECTED loadCornerCardboards : BOOL
VAR_INPUT
	pairIndex : INT;
END_VAR
VAR_OUTPUT
	error : BOOL;
END_VAR
VAR
	errorLeft, errorRight : BOOL;
	leftSuctionArr, rightSuctionArr : POINTER TO SuctionPad;
	leftNextSet, rightNextSet : INT;
	leftMaterial, rightMaterial : STRING;
	leftFold, rightFold : INT;
	
	pair : REFERENCE TO PositionMaterials REF= materialsArr[pairIndex];
	topLeftFold : INT := topLeftFoldsArr[pairIndex];
	topRightFold : INT := topRightFoldsArr[pairIndex];
	bottomLeftFold : INT := bottomLeftFoldsArr[pairIndex];
	bottomRightFold : INT := bottomRightFoldsArr[pairIndex];
END_VAR
{warning disable C0371}

loadCornerCardboards := 
	loadCornerCardboardsEx(
		robot:= robotLeft, 
		aoiLoad:= aoiCornerCardboardLeft, 
		loadStep:= loadStepLeft, 
		pairIndex:= pairIndex, 
		includeTopLeft:= TRUE, 
		includeTopRight:= FALSE, 
		includeBottomLeft:= TRUE, 
		includeBottomRight:= FALSE, 
		error=> errorLeft)
	AND
	loadCornerCardboardsEx(
		robot:= robotRight, 
		aoiLoad:= aoiCornerCardboardRight, 
		loadStep:= loadStepRight, 
		pairIndex:= pairIndex, 
		includeTopLeft:= FALSE, 
		includeTopRight:= TRUE, 
		includeBottomLeft:= FALSE, 
		includeBottomRight:= TRUE, 
		error=> errorLeft);
		
error := errorLeft OR errorRight;

(*
CASE cornerSetLeft OF
	0:
		leftNextSet := Surface.TOP_RIGHT;
		cornerSetLeft := 0;
		
	Surface.TOP_RIGHT: 
		leftNextSet := Surface.TOP_LEFT;
		leftSuctionArr := suctionTopRight;
		leftMaterial := pair.topRight;
		leftFold := topRightFold;
		
	Surface.TOP_LEFT: 
		leftNextSet := Surface.BOTTOM_RIGHT;
		leftSuctionArr := suctionTopLeft;
		leftMaterial := pair.topLeft;
		leftFold := topLeftFold;
		
	Surface.BOTTOM_RIGHT:
		leftNextSet := Surface.BOTTOM_LEFT;
		leftSuctionArr := suctionBottomRight;
		leftMaterial := pair.bottomRight;
		leftFold := bottomRightFold;
		
	Surface.BOTTOM_LEFT: 
		leftNextSet := COMPLETE;
		leftSuctionArr := suctionBottomLeft;
		leftMaterial := pair.bottomLeft;
		leftFold := bottomLeftFold;
END_CASE
IF
	(cornerSetLeft = 0 OR cornerSetLeft = COMPLETE) OR_ELSE
	leftCornerSequence(
		robot:= robotLeft, 
		skid:= skidLeft, 
		suctions := leftSuctionArr,
		loadStep:= loadStepLeft, 
		surfaceID:= cornerSetLeft,
		material:= pair.topRight, 
		foldPos0:= topRightFold, 
		foldPos1:= 0, 
		error=> )
THEN
	cornerSetLeft := leftNextSet;
	loadStepLeft := 0;
END_IF


CASE cornerSetRight OF
	0:
		cornerSetRight := Surface.TOP_RIGHT;
		rightSuctionArr := suctionTopRight;
		
	Surface.TOP_RIGHT:		
		rightNextSet := Surface.BOTTOM_RIGHT;
		rightSuctionArr := suctionTopRight;
		rightMaterial := pair.topRight;
		rightFold := topRightFold;
		
	Surface.BOTTOM_RIGHT: 
		rightNextSet := COMPLETE;
		rightSuctionArr := suctionBottomRight;
		rightMaterial := pair.bottomRight;
		rightFold := bottomRightFold;		
END_CASE
IF
	(cornerSetRight = 0 OR cornerSetRight = COMPLETE) OR_ELSE
	rightCornerSequence(
		robot:= robotRight, 
		skid:= skidRight, 
		suctions := rightSuctionArr,
		loadStep:= loadStepRight, 
		material:= pair.topRight, 
		surfaceID:= cornerSetRight,
		foldPos0:= pair.topRightFold, 
		foldPos1:= 0, 
		error=> )
THEN
	cornerSetRight := rightNextSet;
	loadStepRight := 0;
END_IF



IF cornerSetLeft = COMPLETE AND cornerSetRight = COMPLETE THEN
	loadCornerCardboards := TRUE;
	
	loadStepLeft := loadStepRight := 0;
	cornerSetLeft := cornerSetRight := 0;
END_IF
*)
END_METHOD

METHOD PROTECTED loadCornerCardboardsEx : BOOL
VAR_IN_OUT
	robot : RobotA22;
	aoiLoad : AOI_LoadCornerCardboard;
	loadStep : INT;
END_VAR
VAR_INPUT
	pairIndex : INT;
	includeTopLeft, includeTopRight, includeBottomLeft, includeBottomRight : BOOL;
END_VAR
VAR_OUTPUT
	error : BOOL;
END_VAR
VAR
	suctionsArrLeft, suctionsArrRight : POINTER TO SuctionPad;
	nextSetLeft, nextSetRight : INT;

	pair : REFERENCE TO PositionMaterials REF= materialsArr[pairIndex];
	topLeftFold : INT := topLeftFoldsArr[pairIndex];
	topRightFold : INT := topRightFoldsArr[pairIndex];
	bottomLeftFold : INT := bottomLeftFoldsArr[pairIndex];
	bottomRightFold : INT := bottomRightFoldsArr[pairIndex];
END_VAR
{warning disable C0371}

IF robot.error THEN
	error := TRUE;
	RETURN;
ELSIF robot.reservation <> sectionID AND_THEN NOT robot.reserve(sectionID) THEN
	RETURN;
ELSIF robot.tool <> sectionID AND_THEN NOT robot.changeEOAT(targetTool := sectionID) THEN
	RETURN;
END_IF

error := aoiLoad.error;

CASE loadStep OF
	0:
		loadStep := Surface.BOTTOM_LEFT;
		
	Surface.BOTTOM_LEFT:
		IF NOT includeBottomLeft OR aoiLoad.donePulse THEN
			aoiLoad.execute := FALSE;
			aoiLoad.material := '';
			loadStep := Surface.BOTTOM_RIGHT;
			RETURN;
		END_IF
		
		aoiLoad.surfaceID := loadStep;
		aoiLoad.material := pair.bottomLeft;
		aoiLoad.suctions := suctionBottomLeft;
		aoiLoad.numPads := UPPER_BOUND(suctionBottomLeft, 1) - LOWER_BOUND(suctionBottomLeft, 1) + 1;
		
		aoiLoad.foldPos0 := bottomLeftFold;
		aoiLoad.foldPos1 := 0;
		
		aoiLoad.execute := NOT aoiLoad.busy;
		
	Surface.BOTTOM_RIGHT:
		IF NOT includeBottomRight OR aoiLoad.donePulse THEN
			aoiLoad.execute := FALSE;
			aoiLoad.material := '';
			loadStep := Surface.TOP_LEFT;
			RETURN;
		END_IF
		
		aoiLoad.surfaceID := loadStep;
		aoiLoad.material := pair.bottomRight;
		aoiLoad.suctions := suctionBottomRight;
		aoiLoad.numPads := UPPER_BOUND(suctionBottomRight, 1) - LOWER_BOUND(suctionBottomRight, 1) + 1;
		
		aoiLoad.foldPos0 := bottomRightFold;
		aoiLoad.foldPos1 := 0;
		
		aoiLoad.execute := NOT aoiLoad.busy;
	
	Surface.TOP_LEFT:		
		IF NOT includeTopLeft OR aoiLoad.donePulse THEN
			aoiLoad.execute := FALSE;
			aoiLoad.material := '';
			loadStep := Surface.TOP_RIGHT;
			RETURN;
		END_IF
		
		aoiLoad.surfaceID := loadStep;
		aoiLoad.material := pair.top;
		aoiLoad.suctions := suctionTopLeft;
		aoiLoad.numPads := UPPER_BOUND(suctionTopLeft, 1) - LOWER_BOUND(suctionTopLeft, 1) + 1;
		
		aoiLoad.foldPos0 := topLeftFold;
		aoiLoad.foldPos1 := 0;
		
		aoiLoad.execute := NOT aoiLoad.busy;
		
	Surface.TOP_RIGHT:
		IF NOT includeTopRight OR aoiLoad.donePulse THEN
			aoiLoad.execute := FALSE;
			aoiLoad.material := '';
			loadStep := COMPLETE;
			RETURN;
		END_IF
		
		aoiLoad.surfaceID := loadStep;
		aoiLoad.material := pair.topRight;
		aoiLoad.suctions := suctionTopRight;
		aoiLoad.numPads := UPPER_BOUND(suctionTopRight, 1) - LOWER_BOUND(suctionTopRight, 1) + 1;
		
		aoiLoad.foldPos0 := topRightFold;
		aoiLoad.foldPos1 := 0;
		
		aoiLoad.execute := NOT aoiLoad.busy;
		
	COMPLETE:				
		robot.release(sectionID);
		
		aoiLoad.material := '';
		aoiLoad.execute := FALSE;
		
		loadCornerCardboardsEx := TRUE;
END_CASE
END_METHOD

METHOD loadCornerGuards : BOOL
VAR_INPUT
	pairIndex : INT;
END_VAR
VAR_OUTPUT
	error : BOOL;
END_VAR
VAR
	pair : REFERENCE TO PositionMaterials REF= materialsArr[pairIndex];
	errorLeft, errorRight : BOOL;
END_VAR
{warning disable C0371}

loadCornerGuards := 
	loadCornerGuardsEx(
		robot:= robotLeft, 
		aoiLoad:= aoiCornerGuardLeft, 
		loadStep:= loadStepLeft, 
		pairIndex:= pairIndex, 
		includeTopLeft:= TRUE, 
		includeTopRight:= FALSE, 
		includeBottomLeft:= TRUE, 
		includeBottomRight:= FALSE, 
		error=> errorLeft) 
	AND
	loadCornerGuardsEx(
		robot:= robotRight, 
		aoiLoad:= aoiCornerGuardRight, 
		loadStep:= loadStepRight, 
		pairIndex:= pairIndex, 
		includeTopLeft:= FALSE, 
		includeTopRight:= TRUE, 
		includeBottomLeft:= FALSE, 
		includeBottomRight:= TRUE, 
		error=> errorRight);
		
error := errorLeft OR errorRight;

(*
IF robotLeft.error OR robotRight.error THEN
	error := TRUE;
	RETURN;
	
ELSIF 
	(robotLeft.reservation <> sectionID AND_THEN NOT robotLeft.reserve(sectionID)) OR 
	(robotRight.reservation <> sectionID AND_THEN NOT robotRight.reserve(sectionID))
THEN //loading requires both robots be reserved together
	RETURN;
	
ELSIF //robots have wrong tool
	(robotLeft.tool <> sectionID AND_THEN NOT robotLeft.changeEOAT(targetTool := sectionID)) OR
	(robotRight.tool <> sectionID AND_THEN NOT robotRight.changeEOAT(targetTool := sectionID))
THEN
	RETURN;
	
END_IF

CASE loadStep OF
	0: //top and bottom
		IF aoiCornerGuardLeft.done AND aoiCornerGuardRight.done THEN
			aoiCornerGuardLeft.execute := aoiCornerGuardRight.execute := FALSE;
			aoiCornerGuardLeft.material := aoiCornerGuardRight.material := '';
			loadStep := 10;
			RETURN;
		END_IF
		
		aoiCornerGuardLeft.suctions := 0;
		aoiCornerGuardLeft.surfaceID := Surface.TOP;
		aoiCornerGuardLeft.material := pair.top;
		aoiCornerGuardLeft.numPads := 0;
		
		aoiCornerGuardRight.suctions := suctionBottom;
		aoiCornerGuardRight.surfaceID := Surface.BOTTOM;
		aoiCornerGuardRight.material := pair.bottom;
		aoiCornerGuardRight.numPads := 0;
		
		aoiCornerGuardLeft.execute := NOT aoiCornerGuardLeft.done AND NOT aoiCornerGuardLeft.busy;
		aoiCornerGuardRight.execute := NOT aoiCornerGuardRight.done AND NOT aoiCornerGuardRight.busy;
		
	10: //sides
		IF aoiCornerGuardLeft.done AND aoiCornerGuardRight.done THEN
			aoiCornerGuardLeft.execute := aoiCornerGuardRight.execute := FALSE;
			aoiCornerGuardLeft.material := aoiCornerGuardRight.material := '';
			loadStep := 10;
			RETURN;
		END_IF
		
		aoiCornerGuardLeft.suctions := 0;
		aoiCornerGuardLeft.surfaceID := Surface.LEFT;
		aoiCornerGuardLeft.material := pair.left;
		aoiCornerGuardLeft.numPads := 0;
		
		aoiCornerGuardRight.suctions := 0;
		aoiCornerGuardRight.surfaceID := Surface.RIGHT;
		aoiCornerGuardRight.material := pair.right;
		aoiCornerGuardRight.numPads := 0;
		
		aoiCornerGuardLeft.execute := NOT aoiCornerGuardLeft.done AND NOT aoiCornerGuardLeft.busy;
		aoiCornerGuardRight.execute := NOT aoiCornerGuardRight.done AND NOT aoiCornerGuardRight.busy;
		
	COMPLETE:
		loadStep := 0;
		loadCornerGuards := TRUE;
END_CASE

error := aoiCornerGuardLeft.error OR aoiCornerGuardRight.error;
*)
END_METHOD

METHOD loadCornerGuardsEx : BOOL
VAR_IN_OUT
	robot : RobotA22;
	aoiLoad : AOI_LoadCornerGuard;
	loadStep : INT;
END_VAR
VAR_INPUT
	pairIndex : INT;
	includeTopLeft, includeTopRight, includeBottomLeft, includeBottomRight : BOOL;
END_VAR
VAR_OUTPUT
	error : BOOL;
END_VAR
VAR
	pair : REFERENCE TO PositionMaterials REF= materialsArr[pairIndex];
END_VAR
{warning disable C0371}
IF robot.error THEN
	error := TRUE;
	RETURN;
ELSIF robot.reservation <> sectionID AND_THEN NOT robot.reserve(sectionID) THEN
	RETURN;
ELSIF robot.tool <> sectionID AND_THEN NOT robot.changeEOAT(targetTool := sectionID) THEN
	RETURN;
END_IF

error := aoiLoad.error;

CASE loadStep OF
	0:
		loadStep := Surface.BOTTOM_LEFT;
		
	Surface.BOTTOM_LEFT:
		IF NOT includeBottomLeft OR aoiLoad.donePulse THEN
			aoiLoad.execute := FALSE;
			aoiLoad.material := '';
			loadStep := Surface.BOTTOM_RIGHT;
			RETURN;
		END_IF
		
		aoiLoad.surfaceID := loadStep;
		aoiLoad.material := pair.bottomLeft;
		aoiLoad.suctions := suctionBottomLeft;
		aoiLoad.numPads := UPPER_BOUND(suctionBottomLeft, 1) - LOWER_BOUND(suctionBottomLeft, 1) + 1;
		
		aoiLoad.execute := NOT aoiLoad.busy;
		
	Surface.BOTTOM_RIGHT:
		IF NOT includeBottomRight OR aoiLoad.donePulse THEN
			aoiLoad.execute := FALSE;
			aoiLoad.material := '';
			loadStep := Surface.TOP_LEFT;
			RETURN;
		END_IF
		
		aoiLoad.surfaceID := loadStep;
		aoiLoad.material := pair.bottomRight;
		aoiLoad.suctions := suctionBottomRight;
		aoiLoad.numPads := UPPER_BOUND(suctionBottomRight, 1) - LOWER_BOUND(suctionBottomRight, 1) + 1;
		
		aoiLoad.execute := NOT aoiLoad.busy;
	
	Surface.TOP_LEFT:		
		IF NOT includeTopLeft OR aoiLoad.donePulse THEN
			aoiLoad.execute := FALSE;
			aoiLoad.material := '';
			loadStep := Surface.TOP_RIGHT;
			RETURN;
		END_IF
		
		aoiLoad.surfaceID := loadStep;
		aoiLoad.material := pair.top;
		aoiLoad.suctions := suctionTopLeft;
		aoiLoad.numPads := UPPER_BOUND(suctionTopLeft, 1) - LOWER_BOUND(suctionTopLeft, 1) + 1;
		
		aoiLoad.execute := NOT aoiLoad.busy;
		
	Surface.TOP_RIGHT:
		IF NOT includeTopRight OR aoiLoad.donePulse THEN
			aoiLoad.execute := FALSE;
			aoiLoad.material := '';
			loadStep := COMPLETE;
			RETURN;
		END_IF
		
		aoiLoad.surfaceID := loadStep;
		aoiLoad.material := pair.topRight;
		aoiLoad.suctions := suctionTopRight;
		aoiLoad.numPads := UPPER_BOUND(suctionTopRight, 1) - LOWER_BOUND(suctionTopRight, 1) + 1;
		
		aoiLoad.execute := NOT aoiLoad.busy;
		
	COMPLETE:				
		robot.release(sectionID);
		
		aoiLoad.material := '';
		aoiLoad.execute := FALSE;
		
		loadCornerGuardsEx := TRUE;
END_CASE
END_METHOD

METHOD PROTECTED loadFlatCardboards : BOOL
VAR_INPUT
	pairIndex : INT;
END_VAR
VAR_OUTPUT
	error : BOOL;
END_VAR
VAR
	pair : REFERENCE TO PositionMaterials REF= materialsArr[pairIndex];
	errorLeft, errorRight : BOOL;
END_VAR
{warning disable C0371}

loadFlatCardboards := 
	loadFlatCardboardsEx(
		robot:= robotLeft, 
		aoiLoad:= aoiFlatCardboardLeft, 
		loadStep:= loadStepLeft, 
		pairIndex:= pairIndex, 
		includeTop:= TRUE, 
		includeLeft:= TRUE, 
		includeRight:= FALSE, 
		includeBottom:= FALSE, 
		error=> errorLeft)
	AND
	loadFlatCardboardsEx(
		robot:= robotRight, 
		aoiLoad:= aoiFlatCardboardRight, 
		loadStep:= loadStepRight, 
		pairIndex:= pairIndex, 
		includeTop:= FALSE, 
		includeLeft:= FALSE, 
		includeRight:= TRUE, 
		includeBottom:= TRUE, 
		error=> errorRight);
		
error := errorLeft OR errorRight;

(*
IF robotLeft.error OR robotRight.error THEN
	error := TRUE;
	RETURN;
	
ELSIF 
	(robotLeft.reservation <> sectionID AND_THEN NOT robotLeft.reserve(sectionID)) OR 
	(robotRight.reservation <> sectionID AND_THEN NOT robotRight.reserve(sectionID))
THEN //loading requires both robots be reserved together
	RETURN;
	
ELSIF //robots have wrong tool
	(robotLeft.tool <> sectionID AND_THEN NOT robotLeft.changeEOAT(targetTool := sectionID)) OR
	(robotRight.tool <> sectionID AND_THEN NOT robotRight.changeEOAT(targetTool := sectionID))
THEN
	RETURN;
	
END_IF

CASE loadStep OF
	0: //top and bottom
		IF aoiFlatCardboardLeft.done AND aoiFlatCardboardRight.done THEN
			aoiFlatCardboardLeft.execute := aoiFlatCardboardRight.execute := FALSE;
			aoiFlatCardboardLeft.material := aoiFlatCardboardRight.material := '';
			loadStep := 10;
			RETURN;
		END_IF
		
		aoiFlatCardboardLeft.suctions := 0;
		aoiFlatCardboardLeft.surfaceID := Surface.TOP;
		aoiFlatCardboardLeft.material := pair.top;
		aoiFlatCardboardLeft.numPads := 0;
		
		aoiFlatCardboardRight.suctions := suctionBottom;
		aoiFlatCardboardRight.surfaceID := Surface.BOTTOM;
		aoiFlatCardboardRight.material := pair.bottom;
		aoiFlatCardboardRight.numPads := 0;
		
		aoiFlatCardboardLeft.execute := NOT aoiFlatCardboardLeft.done AND NOT aoiFlatCardboardLeft.busy;
		aoiFlatCardboardRight.execute := NOT aoiFlatCardboardRight.done AND NOT aoiFlatCardboardRight.busy;
		
	10: //sides
		IF aoiFlatCardboardLeft.done AND aoiFlatCardboardRight.done THEN
			aoiFlatCardboardLeft.execute := aoiFlatCardboardRight.execute := FALSE;
			aoiFlatCardboardLeft.material := aoiFlatCardboardRight.material := '';
			loadStep := 10;
			RETURN;
		END_IF
		
		aoiFlatCardboardLeft.suctions := 0;
		aoiFlatCardboardLeft.surfaceID := Surface.LEFT;
		aoiFlatCardboardLeft.material := pair.left;
		aoiFlatCardboardLeft.numPads := 0;
		
		aoiFlatCardboardRight.suctions := 0;
		aoiFlatCardboardRight.surfaceID := Surface.RIGHT;
		aoiFlatCardboardRight.material := pair.right;
		aoiFlatCardboardRight.numPads := 0;
		
		aoiFlatCardboardLeft.execute := NOT aoiFlatCardboardLeft.done AND NOT aoiFlatCardboardLeft.busy;
		aoiFlatCardboardRight.execute := NOT aoiFlatCardboardRight.done AND NOT aoiFlatCardboardRight.busy;
		
	COMPLETE:
		loadStepLeft := loadStepRight := 0;
		loadStep := 0;
		
		loadFlatCardboards := TRUE;
END_CASE

error := aoiFlatCardboardLeft.error OR aoiFlatCardboardRight.error;
*)
END_METHOD

METHOD loadFlatCardboardsEx : BOOL
VAR_IN_OUT
	robot : RobotA22;
	aoiLoad : AOI_LoadFlatCardboard;
	loadStep : INT;
END_VAR
VAR_INPUT
	pairIndex : INT;
	includeTop, includeLeft, includeRight, includeBottom : BOOL;
END_VAR
VAR_OUTPUT
	error : BOOL;
END_VAR
VAR
	pair : REFERENCE TO PositionMaterials REF= materialsArr[pairIndex];
END_VAR
IF robot.error THEN
	error := TRUE;
	RETURN;
ELSIF robot.reservation <> sectionID AND_THEN NOT robot.reserve(sectionID) THEN
	RETURN;
ELSIF robot.tool <> sectionID AND_THEN NOT robot.changeEOAT(targetTool := sectionID) THEN
	RETURN;
END_IF

error := aoiLoad.error;

CASE loadStep OF
	0:
		loadStep := Surface.TOP;
	
	Surface.TOP:	
		IF NOT includeTop OR aoiLoad.donePulse THEN
			aoiLoad.execute := FALSE;
			aoiLoad.material := '';
			loadStep := Surface.BOTTOM;
			RETURN;
		END_IF
		
		aoiLoad.surfaceID := Surface.TOP;
		aoiLoad.material := pair.top;
		aoiLoad.suctions := 0;
		aoiLoad.numPads := 0;
		
		aoiLoad.execute := NOT aoiLoad.busy;
		
	Surface.BOTTOM:
		IF NOT includeBottom OR aoiLoad.donePulse THEN
			aoiLoad.execute := FALSE;
			aoiLoad.material := '';
			loadStep := Surface.LEFT;
			RETURN;
		END_IF
		
		aoiLoad.surfaceID := Surface.BOTTOM;
		aoiLoad.material := pair.bottom;
		aoiLoad.suctions := suctionBottom;
		aoiLoad.numPads := UPPER_BOUND(suctionBottom, 1) - LOWER_BOUND(suctionBottom, 1) + 1;
		
		aoiLoad.execute := NOT aoiLoad.busy;
		
	Surface.LEFT:
		IF NOT includeLeft OR aoiLoad.donePulse THEN
			aoiLoad.execute := FALSE;
			aoiLoad.material := '';
			loadStep := Surface.RIGHT;
			RETURN;
		END_IF
		
		aoiLoad.surfaceID := Surface.LEFT;
		aoiLoad.material := pair.left;
		aoiLoad.suctions := 0;
		aoiLoad.numPads := 0;
		
		aoiLoad.execute := NOT aoiLoad.busy;
		
	Surface.RIGHT:
		IF NOT includeRight OR aoiLoad.donePulse THEN
			aoiLoad.execute := FALSE;
			aoiLoad.material := '';
			loadStep := COMPLETE;
			RETURN;
		END_IF
		
		aoiLoad.surfaceID := Surface.RIGHT;
		aoiLoad.material := pair.right;
		aoiLoad.suctions := 0;
		aoiLoad.numPads := 0;
		
		aoiLoad.execute := NOT aoiLoad.busy;
		
	COMPLETE:				
		robot.release(sectionID);
		
		aoiLoad.material := '';
		aoiLoad.execute := FALSE;
		
		loadFlatCardboardsEx := TRUE;
END_CASE
END_METHOD

METHOD PROTECTED loadLeftCornerCardboards : BOOL
VAR_INPUT
	pair : REFERENCE TO PositionMaterials;
END_VAR
VAR
	suctionsArrLeft, suctionsArrRight : POINTER TO SuctionPad;
	nextSetLeft, nextSetRight : INT;
END_VAR
{warning disable C0371}
(*
CASE cornerSetLeft OF
	0:
		cornerSetLeft := Surface.TOP_RIGHT;
		loadStepLeft := 0;
		
	Surface.TOP_RIGHT: 
		IF
			leftCornerSequence(
				robot:= robotLeft, 
				skid:= skidLeft, 
				suctions := suctionTopRight,
				loadStep:= loadStepLeft, 
				surfaceID:= Surface.TOP_RIGHT,
				material:= pair.topRight, 
				foldPos0:= pair.topRightFold, 
				foldPos1:= 0, 
				error=> )
		THEN
			cornerSetLeft := Surface.TOP_LEFT;
			loadStepLeft := 0;
		END_IF
		
	Surface.TOP_LEFT: 
		IF
			leftCornerSequence(
				robot:= robotLeft, 
				skid:= skidLeft, 
				suctions := suctionTopLeft,
				loadStep:= loadStepLeft, 
				surfaceID:= Surface.TOP_LEFT,
				material:= pair.topLeft, 
				foldPos0:= pair.topLeftFold, 
				foldPos1:= 0, 
				error=> )
		THEN
			cornerSetLeft := Surface.BOTTOM_RIGHT;
			loadStepLeft := 0;
		END_IF
		
	Surface.BOTTOM_RIGHT: 
		IF
			leftCornerSequence(
				robot:= robotLeft, 
				skid:= skidLeft, 
				suctions := suctionBottomRight,
				loadStep:= loadStepLeft, 
				surfaceID:= Surface.BOTTOM_RIGHT,
				material:= pair.bottomRight, 
				foldPos0:= pair.bottomRightFold, 
				foldPos1:= 0, 
				error=> )
		THEN
			cornerSetLeft := Surface.BOTTOM_LEFT;
			loadStepLeft := 0;
		END_IF
		
	Surface.BOTTOM_LEFT: 
		IF
			leftCornerSequence(
				robot:= robotLeft, 
				skid:= skidLeft, 
				suctions := suctionBottomLeft,
				loadStep:= loadStepLeft, 
				surfaceID:= Surface.BOTTOM_LEFT,
				material:= pair.bottomLeft, 
				foldPos0:= pair.bottomLeftFold, 
				foldPos1:= 0, 
				error=> )
		THEN
			cornerSetLeft := COMPLETE;
			loadStepLeft := 0;
		END_IF
END_CASE

//------------------------------------------------------------
IF cornerSetLeft = COMPLETE THEN
	loadStepLeft := 0;
	cornerSetLeft := 0;
	loadLeftCornerCardboards := TRUE;
END_IF
*)
END_METHOD

METHOD PROTECTED loadRightCornerCardboards : BOOL
VAR_INPUT
	pair : REFERENCE TO PositionMaterials;
END_VAR
VAR
	suctionsArrLeft, suctionsArrRight : POINTER TO SuctionPad;
	nextSetLeft, nextSetRight : INT;
END_VAR
(*
{warning disable C0371}
CASE cornerSetRight OF
	0:
		cornerSetRight := Surface.TOP_RIGHT;
		loadStepRight := 0;
		
	Surface.TOP_RIGHT: 
		IF
			rightCornerSequence(
				robot:= robotRight, 
				skid:= skidRight, 
				suctions := suctionTopRight,
				loadStep:= loadStepRight, 
				surfaceID:= Surface.TOP_RIGHT,
				material:= pair.topRight, 
				foldPos0:= pair.topRightFold, 
				foldPos1:= 0, 
				error=> )
		THEN
			cornerSetRight := Surface.BOTTOM_RIGHT;
			loadStepRight := 0;
		END_IF
		
	Surface.BOTTOM_RIGHT: 
		IF
			rightCornerSequence(
				robot:= robotRight, 
				skid:= skidRight, 
				suctions := suctionBottomRight,
				loadStep:= loadStepRight, 
				surfaceID:= Surface.BOTTOM_RIGHT,
				material:= pair.bottomRight, 
				foldPos0:= pair.bottomRightFold, 
				foldPos1:= 0, 
				error=> )
		THEN
			cornerSetRight := Surface.BOTTOM_RIGHT;
			loadStepRight := 0;
		END_IF
		
		cornerSetRight := COMPLETE;			
		loadStepRight := COMPLETE;
		
END_CASE

//------------------------------------------------------------
IF cornerSetRight = COMPLETE THEN	
	loadStepRight := 0;
	cornerSetRight := 0;
	loadRightCornerCardboards := TRUE;
END_IF
*)
END_METHOD

METHOD PROTECTED rightCornerSequence : BOOL
VAR_IN_OUT
	robot : RobotA22;
	skid : SkidMagazine;
	suctions : POINTER TO SuctionPad; //array of SuctionPads, casts from [1..3] to [0..2]
	loadStep : INT;
END_VAR
VAR_INPUT
	surfaceID : Surface;
	material : STRING;
	foldPos0 : INT;
	foldPos1 : INT;
END_VAR
VAR_OUTPUT
	error : BOOL;
END_VAR
VAR
	column : INT;
END_VAR
VAR CONSTANT
	suctionDistance : INT := 10;
END_VAR
(*
{warning disable C0371}
IF material = '' THEN
	rightCornerSequence := TRUE;
	RETURN;
END_IF

CASE loadStep OF
	0:
		robot.clearCommand();
		IF robot.Ready THEN
			loadStep := 10;
		END_IF
		
	10: //overhead to insertion
		IF wrapper.Overhead = '' THEN
			RETURN;
		END_IF
		
		IF robot.eoatDistance < suctionDistance THEN
			robot.HoldMaterial := wrapper.Overhead;
		END_IF
		
	
		IF robot.Done THEN
			loadStep := COMPLETE;
			RETURN;
		END_IF
		
		CASE surfaceID OF
			Surface.TOP_RIGHT:		robot.setGroup(group := 1, value := A22.LOAD_OVERHEAD_TO_UPPER_CORNER);
			Surface.BOTTOM_RIGHT:	robot.setGroup(group := 1, value := A22.LOAD_OVERHEAD_TO_LOWER_CORNER);
		END_CASE
		robot.setGroup(group := 2, value := foldPos0);
		robot.setGroup(group := 3, value := foldPos1);
	
	COMPLETE:
		robot.clearCommand();
		
		CASE surfaceID OF
			Surface.TOP_RIGHT:		suctionTopRight[1].enable := suctionTopRight[3].enable := TRUE;
			Surface.BOTTOM_RIGHT:	suctionBottomRight[1].enable := suctionBottomRight[3].enable := TRUE;
		END_CASE
		
		//suctions[0].enable := TRUE;
		//suctions[2].enable := TRUE;
		
		rightCornerSequence := TRUE;
	
END_CASE
*)
END_METHOD

ACTION stopSequence:
insertionLeft.stop();
insertionRight.stop();
pistonBottom.stop();

robotLeft.clearCommand();
robotRight.clearCommand();
END_ACTION

END_FUNCTION_BLOCK

// ---- DUTs/Machines/FoldingMachine.TcPOU
FUNCTION_BLOCK FoldingMachine
VAR_INPUT CONSTANT
	enable AT %Q* : BOOL;
END_VAR
VAR_OUTPUT
	activeMaterial : STRING;
	
	ready AT %I* : BOOL;
	busy AT %I* : BOOL;
	done AT %I* : BOOL;
	
	//execute AT %Q* : BOOL;
	reset AT %Q* : BOOL;
	foldingPositions AT %Q* : ARRAY[0..1] OF INT;
END_VAR

METHOD setFoldingPositions : BOOL
VAR_INPUT
	foldPos0, foldPos1 : INT;
END_VAR
foldingPositions[0] := foldPos0;
foldingPositions[1] := foldPos1;
END_METHOD

END_FUNCTION_BLOCK

// ---- DUTs/Insertion/Insertion.TcPOU
FUNCTION_BLOCK Insertion //2d insertion that combines a slider (alignment) and screw (push)
VAR_INPUT
	enable : BOOL;
END_VAR
VAR_INPUT //interface references to existing drives
	slider : I_EncodedDrive;
	screw : I_ContinuousDrive;
END_VAR
VAR_OUTPUT
	contact AT %I* : BOOL;
	softContact : BOOL; //temporary
	
	busy : BOOL;
	error : BOOL;
	home : BOOL;
	
	homingComplete : BOOL;
	
	sliderPos : LREAL;
END_VAR
(*
this FB encapsulates 2 drives into a generic insertion machine
the implementation of both drives should be called externally
an Insertion instance should be called in the scope it is declared in
*)

softContact := slider.contact AND screw.contact; //temporary

homingComplete := slider.HomeSet AND screw.HomeSet;

busy := slider.Active OR screw.Active;
error := slider.Error OR screw.Error;
home := slider.AtHome AND screw.AtHome;

sliderPos := slider.CurrentPosition;

METHOD align : BOOL
VAR_INPUT
	targetPos : REAL;
END_VAR
slider.moveAbsolute(newTarget := targetPos);
END_METHOD

METHOD homingSequence : BOOL
VAR_INPUT
END_VAR
IF NOT slider.homeSet THEN
	slider.homingSequence();
END_IF


IF NOT screw.homeSet THEN
	screw.homingSequence();
END_IF

homingSequence := homingComplete;
END_METHOD

METHOD press : BOOL
VAR_INPUT
END_VAR
screw.moveContinuous(direction := MC_Negative_Direction);
END_METHOD

METHOD release : BOOL
VAR_INPUT
END_VAR
screw.moveContinuous(direction := MC_Positive_Direction);
END_METHOD

METHOD reset : BOOL
VAR_INPUT
END_VAR
//slider.reset();
//screw.reset();
END_METHOD

METHOD stop : BOOL
VAR_INPUT
END_VAR
screw.stop();
slider.stop();
END_METHOD

METHOD traverse : BOOL
VAR_INPUT
	direction : MC_Direction;
END_VAR
slider.moveContinuous(direction := MC_Negative_Direction);
END_METHOD

END_FUNCTION_BLOCK

// ---- POUs/A22 - Cardboard-Corner Guard/AOIs/AOI_LoadCornerGuard.TcPOU
FUNCTION_BLOCK AOI_LoadCornerGuard
VAR_INPUT
	execute : BOOL;
END_VAR
VAR_IN_OUT CONSTANT
	sectionID : SectionEnum;
END_VAR
VAR_IN_OUT
	robot : RobotA22;
	magazine : SkidMagazine;
	loadedMaterials : ARRAY[*] OF STRING;
END_VAR
VAR_INPUT
	surfaceID : Surface;
	material : STRING;
	
	suctions : POINTER TO SuctionPad; //access from 0 to numPads-1, not LOWER_BOUND to UPPER_BOUND
	numPads : DINT;
END_VAR
VAR_OUTPUT
	donePulse : BOOL; //this signal turns on 1 cycle after done turns true, should not affect the program structure
	done : BOOL;
	busy : BOOL;
	error : BOOL;
	
	recovery : BOOL;
	failCounter : INT;
END_VAR
VAR
	run : BOOL;
	trigger : R_TRIG;
	doneTrigger : R_TRIG;
	
	column : INT;
	
	suctionTimer : TON;
	step : (IDLE, PREP_ROBOT, GET_FROM_STORAGE, LOAD_TO_INSERTION, COMPLETE, RECOVERY_IDLE, RECOVERY_REMOVE, RECOVERY_LOAD);
	
	i : DINT;
END_VAR
VAR CONSTANT
	suctionDelay : TIME := T#2S;
	suctionDistance : INT := 10;
END_VAR

{warning disable C0371}

trigger(CLK:= execute, Q=> );
doneTrigger(CLK:= done, Q=> donePulse);
busy := trigger.Q OR step > 0;

IF step > IDLE AND_THEN NOT preExecution() THEN //conditions to track before execution
	RETURN;
END_IF

(*
if required bunk was not found on table - restage entire table
if bunk was not loaded correctly - remove bunk, then restage entire table
*)
CASE step OF
	IDLE:
		IF trigger.Q THEN
			recovery := FALSE;
			done := FALSE;
			error := FALSE;
			step := PREP_ROBOT;
		END_IF
		
	PREP_ROBOT:
		robot.clearCommand();
		IF robot.Ready THEN
			step := GET_FROM_STORAGE;
			column := 0;
		END_IF
		
	GET_FROM_STORAGE:		
		IF NOT magazine.findSlot(material := material, index => column) THEN
			error := TRUE;
			RETURN;
		END_IF
		
		IF robot.eoatDistance < suctionDistance THEN //move from table to robot gripper
			robot.HoldMaterial := magazine.getSlot(i := column, error => );
		END_IF
		
		IF robot.Done THEN
			step := COMPLETE;
			RETURN;
		ELSIF robot.materialAtHoldingPosition > 0 THEN
			step := LOAD_TO_INSERTION;
			RETURN;
		END_IF
		
		CASE surfaceID OF
			Surface.TOP_LEFT, Surface.TOP_RIGHT:			robot.setGroup(group := 1, value := A22.LOAD_CORNER_GUARD_UPPER);
			Surface.BOTTOM_LEFT, SURFACE.BOTTOM_RIGHT:		robot.setGroup(group := 1, value := A22.LOAD_CORNER_GUARD_LOWER);
		END_CASE
		robot.setGroup(group := 2, value := column); 
			
	LOAD_TO_INSERTION:
		IF robot.materialAtHoldingPosition > 0 AND robot.HoldMaterial <> '' THEN //move from gripper to insertion
			loadedMaterials[surfaceID] := robot.HoldMaterial;
			robot.HoldMaterial := '';
		END_IF
		
		//numPads/3 <= i < numPads/3 * 2
		FOR i:=(numPads/3)*1 TO (numPads/3)*2-1 BY 1 DO //middle third suctions only
			suctions[i].enable := TRUE;
		END_FOR
		
		IF robot.Done THEN
			suctionTimer.IN := FALSE;
			step := COMPLETE;
			RETURN;
		END_IF
		
		suctionTimer(IN:= , PT:= suctionDelay, Q=> , ET=> );
		suctionTimer.IN := TRUE;
		
		IF suctionTimer.Q THEN
			robot.setGroup(group := 10, value := robot.materialAtHoldingPosition);
		END_IF
	
	COMPLETE:
		robot.clearCommand();
		
		IF //check insertion quality
			SuctionQualityPtrArr(
				suctions := suctions, 
				numPads := numPads, 
				insertionMaterial := loadedMaterials[surfaceID], 
				recipeMaterial := material)
		THEN
			done := TRUE;
			column := 0;
			step := 0;
			
		ELSE //recovery - remove and reload
			failCounter := failCounter + 1;
			step := RECOVERY_IDLE;
		END_IF
		
	//---------RECOVERY-----------------------------------------
	RECOVERY_IDLE:
		robot.clearCommand();
		IF robot.Ready THEN
			step := RECOVERY_REMOVE;
		END_IF
		
	RECOVERY_REMOVE:
		IF robot.Done THEN
			step := RECOVERY_LOAD;
			RETURN;
		END_IF
		
		CASE surfaceID OF
			Surface.TOP_LEFT, Surface.TOP_RIGHT:			robot.setGroup(group := 1, value := A22.REMOVE_CORNER_GUARD_UPPER);
			Surface.BOTTOM_LEFT, SURFACE.BOTTOM_RIGHT:		robot.setGroup(group := 1, value := A22.REMOVE_CORNER_GUARD_LOWER);
		END_CASE
		
	RECOVERY_LOAD:	
		recovery := TRUE;
		error := TRUE;
		
END_CASE

METHOD PRIVATE preExecution : BOOL
VAR_INPUT
END_VAR
{warning disable C0371}
IF material = '' THEN
	done := TRUE;
	RETURN;
END_IF

IF //robot must be ready before execution
	robot.error OR 
	robot.reservation <> sectionID OR 
	robot.tool <> sectionID
THEN
	error := TRUE;
	RETURN;
END_IF

preExecution := TRUE;
END_METHOD

METHOD reset : BOOL
VAR_INPUT
END_VAR
done := FALSE;
busy := FALSE;
error := FALSE;
recovery := FALSE;
failCounter := 0;

column := 0;
step := 0;
END_METHOD

END_FUNCTION_BLOCK

// ---- POUs/A22 - Cardboard-Corner Guard/AOIs/AOI_LoadCornerCardboard.TcPOU
FUNCTION_BLOCK AOI_LoadCornerCardboard
VAR_INPUT
	execute : BOOL;
END_VAR
VAR_IN_OUT CONSTANT
	sectionID : SectionEnum;
END_VAR
VAR_IN_OUT
	robot : RobotA22;
	skid : SkidMagazine;
	loadedMaterials : ARRAY[*] OF STRING;
	overheadTray : STRING;
END_VAR
VAR_INPUT
	surfaceID : Surface;
	material : STRING;
	
	suctions : POINTER TO SuctionPad; //access from 0 to numPads-1, not LOWER_BOUND to UPPER_BOUND
	numPads : DINT;
	
	hasBendingMachine : BOOL;
	foldPos0 : INT;
	foldPos1 : INT;
END_VAR
VAR_OUTPUT
	donePulse : BOOL; //this signal turns on 1 cycle after done turns true and remains on for 1 cycle
	done : BOOL;
	busy : BOOL;
	error : BOOL;
	
	recovery : BOOL;
	failCounter : INT;
END_VAR
VAR
	run : BOOL;
	trigger : R_TRIG;
	doneTrigger : R_TRIG;
	
	column : INT;
	
	suctionTimer : TON;
	
	step : (IDLE, PREP_ROBOT, //common
			GET_FROM_STORAGE, PLACE_TO_OVERHEAD, //left robot only
			GET_FROM_OVERHEAD, //right robot only
			LOAD_TO_INSERTION, COMPLETE, RECOVERY_IDLE, RECOVERY_REMOVE, RECOVERY_LOAD); //common
	
	i : DINT;
END_VAR
VAR CONSTANT
	suctionDelay : TIME := T#2S;
	suctionDistance : INT := 10;
END_VAR

{warning disable C0371}

trigger(CLK:= execute, Q=> );
doneTrigger(CLK:= done, Q=> donePulse);
busy := trigger.Q OR step > 0;

IF step > IDLE AND_THEN NOT preExecution() THEN //conditions to track before execution
	RETURN;
END_IF

CASE step OF
	IDLE:
		IF trigger.Q THEN
			step := PREP_ROBOT;
		END_IF
		
	PREP_ROBOT:
		robot.clearCommand();
		IF robot.Ready THEN
			IF NOT hasBendingMachine THEN //IMPORTANT - this condition differentiates left and right sequences
				step := GET_FROM_STORAGE;
			ELSE
				step := GET_FROM_OVERHEAD;
			END_IF
		END_IF
		
	//----------LEFT ROBOT----------------------------------------
	GET_FROM_STORAGE:
		_GetFromStorage();
	
	PLACE_TO_OVERHEAD:
		_PlaceToOverhead();
	
	//----------RIGHT ROBOT----------------------------------------
	GET_FROM_OVERHEAD:
		_GetFromOverhead();
		
	//----------COMMON----------------------------------------
	LOAD_TO_INSERTION:
		_LoadToInsertion();
		
	COMPLETE:
		robot.clearCommand();

		IF //check insertion quality
			SuctionQualityPtrArr(
				suctions := suctions,
				numPads := numPads, 
				insertionMaterial := loadedMaterials[surfaceID], 
				recipeMaterial := material) 
		THEN
			done := TRUE;
			column := 0;
			step := 0;
			
		ELSE //recovery
			failCounter := failCounter + 1;
			step := RECOVERY_IDLE;
		END_IF
		
	RECOVERY_IDLE:
		robot.clearCommand();
		IF robot.Ready THEN
			step := RECOVERY_REMOVE;
		END_IF
		
	RECOVERY_REMOVE:
		IF robot.Done THEN
			step := RECOVERY_LOAD;
			RETURN;
		END_IF
	
		CASE surfaceID OF
			Surface.TOP_RIGHT:		robot.setGroup(group := 1, value := A22.REMOVE_CARDBOARD_UPPER_CORNER);
			Surface.BOTTOM_RIGHT:	robot.setGroup(group := 1, value := A22.REMOVE_CARDBOARD_LOWER_CORNER);
		END_CASE
		
	RECOVERY_LOAD:
		error := TRUE;
		recovery := TRUE;
			
		IF hasBendingMachine THEN
			step := 0;
		END_IF
		
END_CASE

METHOD PRIVATE _Complete : BOOL
VAR_INPUT
END_VAR
{warning disable C0371}
robot.clearCommand();

IF //check insertion quality
	SuctionQualityPtrArr(
		suctions := suctions,
		numPads := numPads, 
		insertionMaterial := loadedMaterials[surfaceID], 
		recipeMaterial := material) 
THEN
	done := TRUE;
	column := 0;
	step := 0;
	
ELSE //recovery
	failCounter := failCounter + 1;
	step := RECOVERY_IDLE;
END_IF
END_METHOD

METHOD PRIVATE _GetFromOverhead : BOOL
VAR_INPUT
END_VAR
{warning disable C0371}
IF overheadTray = '' AND robot.HoldMaterial = '' THEN
	RETURN;
END_IF

IF robot.eoatDistance < suctionDistance THEN
	robot.HoldMaterial := overheadTray;
	overheadTray := '';
END_IF

IF robot.Done THEN
	step := COMPLETE;
	RETURN;
ELSIF robot.materialAtHoldingPosition > 0 THEN
	step := LOAD_TO_INSERTION;
	RETURN;
END_IF

CASE surfaceID OF
	Surface.TOP_RIGHT:		robot.setGroup(group := 1, value := A22.LOAD_OVERHEAD_TO_UPPER_CORNER);
	Surface.BOTTOM_RIGHT:	robot.setGroup(group := 1, value := A22.LOAD_OVERHEAD_TO_LOWER_CORNER);
END_CASE
robot.setGroup(group := 2, value := 0);
robot.setGroup(group := 3, value := 0);
END_METHOD

METHOD PRIVATE _GetFromStorage : BOOL
VAR_INPUT
END_VAR
{warning disable C0371}
IF NOT skid.findSlot(material := material, index=> column) THEN
	error := TRUE;
	RETURN;
END_IF

IF robot.eoatDistance < suctionDistance THEN
	robot.HoldMaterial := skid.getSlot(i := column);
END_IF

IF robot.Done THEN
	
	CASE surfaceID OF //determine what to do with the cardboard - load to insertion or move to overhead tray
		Surface.TOP_RIGHT, Surface.BOTTOM_RIGHT:	step := PLACE_TO_OVERHEAD;
		Surface.TOP_LEFT, Surface.BOTTOM_LEFT:		step := LOAD_TO_INSERTION;
	END_CASE
	
	RETURN;
END_IF

robot.setGroup(group := 1, value := A22.TRANSFER_TO_BENDER);
robot.setGroup(group := 2, value := foldPos0);
robot.setGroup(group := 3, value := foldPos1);
END_METHOD

METHOD PRIVATE _LoadToInsertion : BOOL
VAR_INPUT
END_VAR
{warning disable C0371}
FOR i:=(numPads/3)*0 TO (numPads/3)*1 - 1 BY 1 DO //first third suctions only
	suctions[i].enable := TRUE;
END_FOR

FOR i:=(numPads/3)*2 TO (numPads/3)*3 - 1 BY 1 DO //last third suctions only
	suctions[i].enable := TRUE;
END_FOR

IF robot.Done THEN
	suctionTimer.IN := FALSE;
	step := COMPLETE;
	RETURN;
END_IF

suctionTimer(IN:= , PT:= suctionDelay, Q=> , ET=> );
suctionTimer.IN := TRUE;

IF suctionTimer.Q THEN
	robot.setGroup(group := 10, value := robot.materialAtHoldingPosition);
END_IF
END_METHOD

METHOD PRIVATE _PlaceToOverhead : BOOL
VAR_INPUT
END_VAR
{warning disable C0371}
IF robot.Done THEN
	step := COMPLETE;
	RETURN;
END_IF

robot.setGroup(group := 1, value := A22.TRANSFER_TO_OVERHEAD);
robot.setGroup(group := 2, value := 0);
robot.setGroup(group := 3, value := 0);
END_METHOD

METHOD PRIVATE preExecution : BOOL
VAR_INPUT
END_VAR
{warning disable C0371}
IF material = '' THEN
	done := TRUE;
	RETURN;
END_IF

IF //robot must be ready before execution
	robot.error OR 
	robot.reservation <> sectionID OR 
	robot.tool <> sectionID
THEN
	error := TRUE;
	RETURN;
END_IF

preExecution := TRUE;
END_METHOD

METHOD reset : BOOL
VAR_INPUT
END_VAR
done := FALSE;
busy := FALSE;
error := FALSE;
recovery := FALSE;
failCounter := 0;

column := 0;
step := 0;
END_METHOD

END_FUNCTION_BLOCK

// ---- POUs/A22 - Cardboard-Corner Guard/AOIs/AOI_LoadFlatCardboard.TcPOU
FUNCTION_BLOCK AOI_LoadFlatCardboard
VAR_INPUT
	execute : BOOL;
END_VAR
VAR_IN_OUT CONSTANT
	sectionID : SectionEnum;
END_VAR
VAR_IN_OUT
	robot : RobotA22;
	skid : SkidMagazine;
	loadedMaterials : ARRAY[*] OF STRING;
END_VAR
VAR_INPUT
	surfaceID : Surface;
	material : STRING;
	
	suctions : POINTER TO SuctionPad; //access from 0 to numPads-1, not LOWER_BOUND to UPPER_BOUND
	numPads : DINT;
END_VAR
VAR_OUTPUT
	donePulse : BOOL;
	done : BOOL;
	busy : BOOL;
	error : BOOL;
	
	recovery : BOOL;
	failCounter : INT;
END_VAR
VAR
	run : BOOL;
	trigger : R_TRIG;
	doneTrigger : R_TRIG;
	
	column : INT;
	
	suctionTimer : TON;
	step : (IDLE, PREP_ROBOT, GET_FROM_STORAGE, LOAD_TO_INSERTION, COMPLETE, RECOVERY_IDLE, RECOVERY_REMOVE, RECOVERY_WAIT, RECOVERY_LOAD);
	
	i : DINT;
END_VAR
VAR_STAT CONSTANT
	suctionDelay : TIME := T#2S;
	suctionDistance : INT := 10;
END_VAR

{warning disable C0371}

trigger(CLK:= execute, Q=> );
doneTrigger(CLK:= done, Q=> donePulse);
busy := trigger.Q OR step > 0;

IF step > IDLE AND_THEN NOT preExecution() THEN //conditions to track before execution
	RETURN;
END_IF

(*
if bunk was not loaded correctly - remove bunk, then restage entire table
*)
CASE step OF
	IDLE:
		IF trigger.Q THEN
			recovery := FALSE;
			done := FALSE;
			error := FALSE;
			step := PREP_ROBOT;
		END_IF
		
	PREP_ROBOT:
		robot.clearCommand();
		IF robot.Ready THEN
			step := GET_FROM_STORAGE;
			column := 0;
		END_IF
		
	GET_FROM_STORAGE:		
		IF NOT skid.findSlot(material := material, index => column) THEN
			error := TRUE;
			RETURN;
		END_IF
		
		IF robot.eoatDistance < suctionDistance THEN//move from table to robot gripper
			robot.HoldMaterial := skid.getSlot(i := column, error => );;
		END_IF
		
		IF robot.Done THEN
			step := COMPLETE;
			RETURN;
		ELSIF robot.materialAtHoldingPosition >= 1 AND robot.materialAtHoldingPosition <= 8 THEN
			step := LOAD_TO_INSERTION;
			RETURN;
		END_IF
		
		CASE surfaceID OF
			Surface.TOP_LEFT, Surface.TOP_RIGHT:			robot.setGroup(group := 1, value := A22.LOAD_CORNER_GUARD_UPPER);
			Surface.BOTTOM_LEFT, SURFACE.BOTTOM_RIGHT:		robot.setGroup(group := 1, value := A22.LOAD_CORNER_GUARD_LOWER);
		END_CASE
		robot.setGroup(group := 2, value := column); 
			
	LOAD_TO_INSERTION:
		IF robot.materialAtHoldingPosition > 0 AND robot.HoldMaterial <> '' THEN //move from gripper to insertion
			loadedMaterials[surfaceID] := robot.HoldMaterial;
			robot.HoldMaterial := '';
		END_IF
		
		//only bottom cardboard uses suction
		CASE surfaceID OF
			Surface.BOTTOM:		SetSuctionsPtrArr(suctions := suctions, numPads := numPads, state := TRUE);
		END_CASE
		
		IF robot.Done THEN
			suctionTimer.IN := FALSE;
			step := COMPLETE;
			RETURN;
		END_IF
		
		suctionTimer(IN:= , PT:= suctionDelay, Q=> , ET=> );
		suctionTimer.IN := TRUE;
		
		IF suctionTimer.Q THEN
			robot.setGroup(group := 10, value := robot.materialAtHoldingPosition);
		END_IF
	
	COMPLETE:
		robot.clearCommand();
		
		IF //if bottom then check insertion, otherwise done
			surfaceID <> Surface.BOTTOM OR_ELSE 
			SuctionQualityPtrArr(
				suctions := suctions, 
				numPads := numPads, 
				insertionMaterial := loadedMaterials[surfaceID], 
				recipeMaterial := material)
		THEN
			done := TRUE;
			column := 0;
			step := 0;
			
		ELSE //recovery - remove and reload
			failCounter := failCounter + 1;
			step := RECOVERY_IDLE;
		END_IF
		
	//---------RECOVERY-----------------------------------------
	RECOVERY_IDLE:
		robot.clearCommand();
		IF robot.Ready THEN
			step := RECOVERY_REMOVE;
		END_IF
		
	RECOVERY_REMOVE:
		IF robot.Done THEN
			step := RECOVERY_LOAD;
			RETURN;
		END_IF
		
		CASE surfaceID OF
			Surface.BOTTOM:		robot.setGroup(group := 1, value := A22.REMOVE_CARDBOARD_BOTTOM);
		END_CASE
		
	RECOVERY_LOAD:	
		recovery := TRUE;
		error := TRUE;
		
END_CASE

METHOD PRIVATE preExecution : BOOL
VAR_INPUT
END_VAR
{warning disable C0371}
IF material = '' THEN
	done := TRUE;
	RETURN;
END_IF

IF //robot must be ready before execution
	robot.error OR 
	robot.reservation <> sectionID OR 
	robot.tool <> sectionID
THEN
	error := TRUE;
	RETURN;
END_IF

preExecution := TRUE;
END_METHOD

METHOD reset : BOOL
VAR_INPUT
END_VAR
done := FALSE;
busy := FALSE;
error := FALSE;
recovery := FALSE;
failCounter := 0;

column := 0;
step := 0;
END_METHOD

END_FUNCTION_BLOCK

// ---- POUs/Hardware Calls/SetSuctions.TcPOU
FUNCTION SetSuctions : BOOL
VAR_IN_OUT
	suctions : ARRAY[*] OF SuctionPad;
END_VAR
VAR_INPUT
	state : BOOL;
END_VAR
VAR
	i : DINT;
END_VAR

FOR i:=LOWER_BOUND(suctions, 1) TO UPPER_BOUND(suctions, 1) BY 1 DO
	suctions[i].enable := state;
END_FOR

END_FUNCTION

// ---- POUs/Materials/MatchesMaterialType.TcPOU
FUNCTION MatchesMaterialType : BOOL
VAR_INPUT
	pair : REFERENCE TO PositionMaterials;
	materialType : STRING;
END_VAR
VAR
END_VAR

MatchesMaterialType :=
	FIND(pair.top, materialType) > 0 OR
	FIND(pair.left, materialType) > 0 OR
	FIND(pair.right, materialType) > 0 OR
	FIND(pair.bottom, materialType) > 0 OR
	
	FIND(pair.topLeft, materialType) > 0 OR
	FIND(pair.topRight, materialType) > 0 OR
	FIND(pair.bottomLeft, materialType) > 0 OR
	FIND(pair.bottomRight, materialType) > 0 ;

END_FUNCTION

// ---- POUs/Hardware Calls/CallHardwareModules.TcPOU
FUNCTION CallHardwareModules : BOOL //only purpose of this function is to call modules from Hardware

robot3();
robot4();

skidA22Left(slots := skidHmiA22Left);
skidA22Right(slots := skidHmiA22Right);

magazineA22Left(slots := magazineHmiA22Left);
magazineA22Right(slots := magazineHmiA22Right);

wrapperA22();
benderA22Left();

horizontalDriveA22Left();
horizontalDriveA22Right();

verticalDriveA22Left();
verticalDriveA22Right();

pistonA22Bottom();

insertionA22Left(
	enable:= TRUE, 
	slider:= verticalDriveA22Left, 
	screw:= horizontalDriveA22Left, 
	contact=> , 
	softContact=> , 
	busy=> , 
	error=> , 
	home=> , 
	homingComplete=> , 
	sliderPos=> );
	
insertionA22Right(
	enable:= TRUE, 
	slider:= verticalDriveA22Right, 
	screw:= horizontalDriveA22Right, 
	contact=> , 
	softContact=> , 
	busy=> , 
	error=> , 
	home=> , 
	homingComplete=> , 
	sliderPos=> );

END_FUNCTION

// ---- DUTs/Insertion/Drives/ServoNC.TcPOU
FUNCTION_BLOCK ServoNC EXTENDS FBA_Drive IMPLEMENTS I_EncodedDrive
VAR_OUTPUT	
	ready : BOOL;
	position : LREAL;
	velocity : LREAL;
END_VAR
VAR
	axis : AXIS_REF;
	
	mcReadPosition : MC_ReadActualPosition;
	mcReadVelocity : MC_ReadActualVelocity;
	mcReadError : MC_ReadAxisError;
	mcReset : MC_Reset;
	
	mcPower : MC_Power;
	mcMoveAbsolute : MC_MoveAbsolute;
	mcMoveRelative : MC_MoveRelative;
	mcMoveVelocity : MC_MoveVelocity;
	
	mcSetPosition : MC_SetPosition;
	mcStop : MC_Stop;
END_VAR
VAR_STAT CONSTANT
	targetingVelocity : INT := 500;
	continuousVelocity : INT := 100;
END_VAR

override();

blocks();

mcReset.Execute := FALSE;
mcMoveAbsolute.Execute := FALSE;
mcMoveRelative.Execute := FALSE;
mcMoveVelocity.Execute := FALSE;
mcSetPosition.Execute := FALSE;
mcStop.Execute := FALSE;

blocks();

ready := bEnable AND NOT Active AND HomeSet;

PROPERTY Active : BOOL
GET
Active := 
	mcMoveAbsolute.Busy OR 
	mcMoveRelative.Busy OR 
	mcMoveVelocity.Busy OR 
	mcSetPosition.Busy OR 
	mcReset.Busy OR 
	mcStop.Busy OR 
	step <> 0;
END_GET
END_PROPERTY

METHOD PRIVATE blocks : BOOL
mcReadPosition(
	Axis:= axis, 
	Enable:= TRUE, 
	Valid=> , 
	Busy=> , 
	Error=> , 
	ErrorID=> , 
	Position=> position);
	
mcReadVelocity(
	Axis:= axis, 
	Enable:= TRUE, 
	Valid=> , 
	Busy=> , 
	Error=> , 
	ErrorID=> , 
	ActualVelocity=> velocity);
	
mcReadError(
	Axis:= axis, 
	Enable:= TRUE, 
	Valid=> , 
	Busy=> , 
	Error=> , 
	ErrorID=> , 
	AxisErrorID=> );

mcReset(
	Axis:= axis, 
	Execute:= , 
	Done=> , 
	Busy=> , 
	Error=> , 
	ErrorID=> );

mcPower(
	Axis:= axis, 
	Enable:= bEnable, 
	Enable_Positive:= TRUE, 
	Enable_Negative:= TRUE, 
	Override:= 100, 
	BufferMode:= , 
	Options:= , 
	Status=> , 
	Busy=> , 
	Active=> , 
	Error=> , 
	ErrorID=> );

mcMoveAbsolute(
	Axis:= axis, 
	Execute:= , 
	Position:= , 
	Velocity:= targetingVelocity, 
	Acceleration:= , 
	Deceleration:= , 
	Jerk:= , 
	BufferMode:= , 
	Options:= , 
	Done=> , 
	Busy=> , 
	Active=> , 
	CommandAborted=> , 
	Error=> , 
	ErrorID=> );
	
mcMoveRelative(
	Axis:= axis, 
	Execute:= , 
	Distance:= ,
	Velocity:= targetingVelocity, 
	Acceleration:= , 
	Deceleration:= , 
	Jerk:= , 
	BufferMode:= , 
	Options:= , 
	Done=> , 
	Busy=> , 
	Active=> , 
	CommandAborted=> , 
	Error=> , 
	ErrorID=> );
	
mcMoveVelocity( //stopped with stop();
	Axis:= axis, 
	Execute:= , 
	Velocity:= continuousVelocity, 
	Acceleration:= , 
	Deceleration:= , 
	Jerk:= , 
	Direction:= , 
	BufferMode:= , 
	Options:= , 
	InVelocity=> , 
	Busy=> , 
	Active=> , 
	CommandAborted=> , 
	Error=> , 
	ErrorID=> );
	
mcSetPosition(
	Axis:= axis, 
	Execute:= , 
	Position:= , 
	Mode:= , 
	Options:= , 
	Done=> , 
	Busy=> , 
	Error=> , 
	ErrorID=> );
	
mcStop(
	Axis:= axis, 
	Execute:= , 
	Deceleration:= , 
	Jerk:= , 
	Options:= , 
	Done=> , 
	Busy=> , 
	Active=> , 
	CommandAborted=> , 
	Error=> , 
	ErrorID=> );
END_METHOD

PROPERTY CurrentPosition : LREAL
GET
CurrentPosition := position;
END_GET
SET
position := CurrentPosition;
END_SET
END_PROPERTY

PROPERTY Error : BOOL
GET
error := 
	mcMoveAbsolute.Error OR 
	mcMoveRelative.Error OR 
	mcMoveVelocity.Error OR 
	mcSetPosition.Error OR 
	mcReset.Error OR 
	mcStop.Error OR
	mcReadError.AxisErrorID > 0;
END_GET
END_PROPERTY

METHOD homingSequence : BOOL
CASE step OF
	Homing.IDLE:
		reset();
		IF bEnable THEN
			step := Homing.START;
		END_IF
		
	Homing.START:
		IF AtHome THEN
			mcMoveVelocity.Execute := FALSE;
			step := Homing.STOP;
			
		ELSIF AtInnerLimit THEN
			mcMoveVelocity.Execute := FALSE;
			step := Homing.RETRY;
			
		ELSE
			mcMoveVelocity.Direction := MC_Negative_Direction;
			mcMoveVelocity.Execute := NOT mcMoveVelocity.Execute;
		END_IF
		
	Homing.RETRY:
		IF AtOuterLimit THEN
			mcMoveVelocity.Execute := FALSE;
			step := Homing.START;
		ELSE
			mcMoveVelocity.Direction := MC_Positive_Direction;
			mcMoveVelocity.Execute := NOT mcMoveVelocity.Execute;
		END_IF
		
	Homing.STOP:
		IF velocity = 0 THEN
			mcStop.Execute := FALSE;
			step := Homing.SET;
			RETURN;
		END_IF
		
		mcStop.Execute := TRUE;
		
	Homing.SET:
		IF position = 0 THEN
			mcSetPosition.Execute := FALSE;
			homingSequence := TRUE;
			step := Homing.DONE;
			RETURN;
		END_IF
		
		mcSetPosition.Position := 0;
		mcSetPosition.Execute := TRUE;
		
	Homing.DONE:
		homingComplete := TRUE;
		step := Homing.IDLE;
		
END_CASE
END_METHOD

METHOD moveAbsolute : BOOL
VAR_INPUT
	newTarget : LREAL;
END_VAR
(*
VAR_OUTPUT
	fault : BOOL;
END_VAR
*)
IF NOT Active AND NOT error THEN
	mcMoveAbsolute.Position := newTarget;
	mcMoveAbsolute.Execute := TRUE;
END_IF

moveAbsolute := (*mcMoveAbsolute.Done AND mcMoveAbsolute.Active;*)
	position = newTarget;
END_METHOD

METHOD moveContinuous : BOOL
VAR_INPUT
	//direction : BOOL; //direction (F = inwards, T = outwards)
	direction : MC_Direction;
END_VAR
(*
IF mcMoveVelocity.Active THEN
	stop();
END_IF

IF NOT mcStop.Done THEN
	RETURN;
END_IF
*)
(*
IF direction THEN
	mcMoveVelocity.Direction := MC_Positive_Direction;
ELSE
	mcMoveVelocity.Direction := MC_Negative_Direction;
END_IF
*)
mcMoveVelocity.Direction := direction;

IF NOT mcMoveVelocity.Error THEN
	mcMoveVelocity.Execute := TRUE;
	moveContinuous := TRUE;
END_IF
END_METHOD

METHOD moveRelative : BOOL
VAR_INPUT
	distance : LREAL;
END_VAR
mcMoveRelative.Distance := distance;

moveRelative := mcMoveRelative.Done;
END_METHOD

METHOD PRIVATE override : BOOL
VAR_INPUT
END_VAR
(*
-at home and attempting to traverse outward
-at outer limit and attempting to traverse outward
-at inner limit and attempting to traverse inwards
*)
(*
inward = negative direction, negative velocity
outward = positive direction, positive velocity
*)

IF error THEN
	stop();
	reset();
	
ELSIF
	AtHome AND (TargetPosition > CurrentPosition OR velocity > 0) OR
	AtOuterLimit AND (TargetPosition > CurrentPosition OR velocity > 0) OR
	AtInnerLimit AND (TargetPosition < CurrentPosition OR velocity < 0)
THEN
	stop();
END_IF
END_METHOD

METHOD reset : BOOL
VAR_INPUT
END_VAR
mcReset.Execute := TRUE;

reset := mcReset.Done;
END_METHOD

METHOD stop : BOOL
VAR_INPUT
END_VAR
mcStop.Execute := TRUE;

mcMoveAbsolute.Execute := FALSE;
mcMoveRelative.Execute := FALSE;
mcMoveVelocity.Execute := FALSE;
END_METHOD

PROPERTY TargetPosition : LREAL
GET
END_GET
SET
moveAbsolute(newTarget := TargetPosition);
END_SET
END_PROPERTY

METHOD toHome : BOOL
VAR_INPUT
END_VAR
moveAbsolute(newTarget := 0);

toHome := AtHome;
END_METHOD

END_FUNCTION_BLOCK

// ---- DUTs/Insertion/ABSTRACT/FBA_Drive.TcPOU
FUNCTION_BLOCK ABSTRACT FBA_Drive IMPLEMENTS I_Drive
VAR_INPUT
	bEnable : BOOL;
END_VAR
VAR //constructor
	limitSensorDefaultState : BOOL;
	//when a traverse sensor is opposite of this value, the respective property becomes TRUE
	//all sensors for a drive should be of the same type - do not mix & match PNP and NPN sensors on the same drive
END_VAR
VAR
	contactSensor AT %I* : BOOL;
	
	outerLimit AT %I* : BOOL; //replacable with traverseLimit
	innerLimit AT %I* : BOOL; //replacable with homeLimit
	home AT %I* : BOOL;
	
	homingComplete : BOOL;
	
	step : Homing;
END_VAR
(*
this abstract FB only specifies the minimum data for any drive/servo
*)

{attribute 'monitoring':='call'}
PROPERTY ABSTRACT Active : BOOL
GET
END_GET
END_PROPERTY

{attribute 'monitoring':='call'}
PROPERTY AtHome : BOOL
GET
AtHome := home <> limitSensorDefaultState;
END_GET
END_PROPERTY

{attribute 'monitoring':='call'}
PROPERTY AtInnerLimit : BOOL
GET
AtInnerLimit := innerLimit <> limitSensorDefaultState;
END_GET
END_PROPERTY

{attribute 'monitoring':='call'}
PROPERTY AtOuterLimit : BOOL
GET
AtOuterLimit := outerLimit <> limitSensorDefaultState;
END_GET
END_PROPERTY

{attribute 'monitoring':='call'}
PROPERTY Contact : BOOL
GET
Contact := contactSensor;
END_GET
END_PROPERTY

{attribute 'monitoring':='call'}
PROPERTY ABSTRACT Error : BOOL
GET
END_GET
END_PROPERTY

{attribute 'monitoring':='call'}
PROPERTY HomeSet : BOOL
GET
HomeSet := homingComplete;
END_GET
END_PROPERTY

METHOD ABSTRACT homingSequence : BOOL
VAR_INPUT
END_VAR
END_METHOD

METHOD ABSTRACT reset : BOOL
VAR_INPUT
END_VAR
END_METHOD

METHOD ABSTRACT stop : BOOL
VAR_INPUT
END_VAR
END_METHOD

END_FUNCTION_BLOCK

// ---- DUTs/Insertion/Drives/ClearLinkMC.TcPOU
FUNCTION_BLOCK ClearLinkMC EXTENDS FBA_Drive IMPLEMENTS I_EncodedDrive //I_PositionalDrive, I_ContinuousDrive
VAR_OUTPUT
	pulse AT %Q* : INT; //num pulses
	brakeRelease AT %Q* : BOOL;
	enable : BOOL;
	A : BOOL; //direction (T = outwards, F = inwards)
	B : BOOL; //home bit
	clear : BOOL; //reset bit
	
	hlfb AT %I* : REAL := -9999; //high level feedback, if -9999 then servo is idle
END_VAR
VAR //constructor
	homingDirection : BOOL; //homing direction (F = inwards, T = outwards)
	minPosition : LREAL;
	displacementPerRotation : LREAL; //displacement per revolution	
	unitsPerPulse : INT := 800; //800 Teknic units per revolution
END_VAR
VAR	
	outputRegister AT %Q* : INT;
	pulseRequest : INT;
	
	pulsePosition : INT;
	pulseCounter : INT;
	
	retryHoming : TON;
	homingDelay : TON;
	resetPulse : TP;
	
	mode : (HOLD, TARGET, CONTINUOUS, RESET_ERR);
	calculation : (IDLE, DOWN, UP, CALCULATE, DONE);
	
	maxPosition : LREAL;
	position, targetPos : LREAL;
END_VAR
VAR
	rotationsPerPulse : INT; //revolutions per pulse
	displacementPerPulse : LREAL; //displacement per pulse
END_VAR
VAR_STAT CONSTANT
	resetWidth : TIME := T#1000MS;
	delayWidth : TIME := T#200MS;
END_VAR

//M-connector output register
outputRegister.0 := enable AND bEnable; 	//enable
outputRegister.1 := A; 						//direction bit
outputRegister.2 := B; 						//homing bit - after startup, set to TRUE to begin homing, then set to FALSE to finish homing
outputRegister.3 := clear; 					//reset bit

rotationsPerPulse := unitsPerPulse/800; //Teknic constant - 800 units per rotation
displacementPerPulse := displacementPerRotation * rotationsPerPulse;

resetPulse(IN:= , PT:= resetWidth, Q=> clear, ET=> ); //reset pulse

IF NOT bEnable THEN
	homingComplete := FALSE;
	mode := HOLD;
END_IF

override();

CASE mode OF		
	HOLD: //hold current position, no motion
		pulse := 0;
		pulseRequest := 0;
	
	TARGET:	//target a given position
		IF WithinTolerance(position, targetPos, displacementPerPulse) THEN
			pulseRequest := 0;
			mode := HOLD;
			
		ELSIF NOT Active THEN
			A :=  position < targetPos;
			(*
			2 options to traverse to a target position:
				a)  send all pulses at once - single continuous motion but may exceed limits
				b)  1 pulse at a time - choppy but safer
			*)
			//pulseRequest := TO_INT(ABS(position - targetPos)/distancePerPulse);
			pulseRequest := 1;
			
		END_IF
		
	CONTINUOUS: //single pulses in the direction specified by moveContinuous()
		pulseRequest := 1;
		
	RESET_ERR: //reset pulse, servo may need to be rehomed aftewards
		pulse := 0;
		pulseRequest := 0;
		resetPulse.IN := TRUE;
		
		IF resetPulse.Q THEN
			resetPulse.IN := FALSE;
			mode := HOLD;
		END_IF
		
END_CASE

sequence();

PROPERTY Active : BOOL
GET
Active := hlfb <> -9999;
END_GET
END_PROPERTY

METHOD PRIVATE calculatePositions : BOOL
(*
the purpose of this method is calculate the position at the outer limit

complete a full range traverse while counting the pulses, then multiply
	displacement per rotation
	rotations per pulse
	number of pulses for the traversal
and add to position at inner limit to get position at outer limit
*)
CASE calculation OF
	IDLE:
		calculation := DOWN;
		
	DOWN:
		moveContinuous(direction := MC_Negative_Direction);
		
		IF AtInnerLimit THEN
			calculation := UP;
			pulseCounter := 0;
		END_IF
		
	UP:
		moveContinuous(direction := MC_Positive_Direction);
		
		IF AtHome THEN
			maxPosition := minPosition + (displacementPerRotation * rotationsPerPulse * pulseCounter);
			calculation := DONE;
		END_IF
		
	DONE:
		calculatePositions := TRUE;
		
END_CASE
END_METHOD

PROPERTY CurrentPosition : LREAL
GET
CurrentPosition := position;
END_GET
SET
position := CurrentPosition;
END_SET
END_PROPERTY

PROPERTY Error : BOOL
GET
END_GET
END_PROPERTY

METHOD homingSequence : BOOL
retryHoming(IN:= , PT:= resetWidth, Q=> , ET=> );
homingDelay(IN:= , PT:= delayWidth, Q=> , ET=> );

CASE step OF
	Homing.IDLE:
		enable := FALSE;
		A := FALSE;
		B := FALSE;
		brakeRelease := TRUE;
		
		homingComplete := FALSE;
		step := Homing.START;
		
	Homing.START:
		IF homingDelay.Q THEN
			homingDelay.IN := FALSE;
			step := Homing.SET;
			
		ELSIF AtHome THEN
			homingDelay.IN := TRUE;
			
		ELSIF AtOuterLimit THEN
			step := Homing.RETRY;
		
		ELSE
			enable := TRUE;
			A := FALSE;
			B := TRUE;
			brakeRelease := TRUE;
		
		END_IF
	
	Homing.RETRY:
		IF AtInnerLimit THEN
			retryHoming.IN := TRUE;
			enable := FALSE;
			
			IF retryHoming.Q THEN
				retryHoming.IN := FALSE;
				step := Homing.START;
			END_IF
			
		ELSE
			enable := TRUE;
			A := FALSE;
			B := FALSE;
			brakeRelease := TRUE;
			
			mode := CONTINUOUS;
		END_IF

	Homing.SET:
		enable := TRUE;
		A := FALSE;
		B := FALSE;
		brakeRelease := TRUE;
		
		IF calculatePositions() THEN
			step := Homing.DONE;
		END_IF
		
	Homing.DONE:
		homingSequence := homingComplete := TRUE;
		
		mode := HOLD;
		step := Homing.IDLE;
	
END_CASE
END_METHOD

METHOD moveAbsolute : BOOL
VAR_INPUT
	newTarget : LREAL;
END_VAR
(*
IF homingDirection THEN //homing is outwards
	targetPos := maxPosition - newTarget;
	
ELSE //homing is inwards
	targetPos := newTarget;
END_IF
*)

targetPos := newTarget;
mode := TARGET;
END_METHOD

METHOD moveContinuous : BOOL
VAR_INPUT
	direction : MC_Direction;
END_VAR
IF direction = MC_Negative_Direction THEN
	A := FALSE;
ELSIF direction = MC_Positive_Direction THEN
	A := TRUE;
END_IF

mode := CONTINUOUS;
END_METHOD

METHOD moveRelative : BOOL
VAR_INPUT
	distance : LREAL;
END_VAR
targetPos := targetPos + distance;

mode := TARGET;
END_METHOD

METHOD PRIVATE override : BOOL
VAR_INPUT
END_VAR
(*
allowable motion is between AtHome and AtInnerLimit
*)
IF
	(AtHome AND A) OR
	(AtOuterLimit AND A) OR
	(AtInnerLimit AND NOT A)
THEN
	mode := HOLD;
END_IF

//--------------------
IF AtHome THEN
	IF homingDirection THEN //homing is outwards
		position := maxPosition;
	ELSE
		position := minPosition;
	END_IF
END_IF
END_METHOD

METHOD reset : BOOL
VAR_INPUT
END_VAR
mode := RESET_ERR;
END_METHOD

METHOD PRIVATE sequence : BOOL
VAR_INPUT
END_VAR
IF Active THEN //servo is active
	IF A THEN //positive direction
		position := position + (displacementPerPulse * pulse);
		pulsePosition := pulsePosition + pulse;
		
		pulseCounter := pulseCounter + pulse;
	ELSE //negative direction
		position := position - (displacementPerPulse * pulse);
		pulsePosition := pulsePosition - pulse;
		
		pulseCounter := pulseCounter - pulse;
	END_IF
	pulse := 0; //pulses already received, can be set to 0 so position change is not compounded

ELSIF pulse = 0 THEN //servo is not active
	pulse := pulseRequest;
	
END_IF
END_METHOD

METHOD stop : BOOL
VAR_INPUT
END_VAR
mode := HOLD;
END_METHOD

PROPERTY TargetPosition : LREAL
GET
END_GET
SET
targetPos := TargetPosition;
END_SET
END_PROPERTY

END_FUNCTION_BLOCK

// ---- POUs/FB_System.TcPOU
FUNCTION_BLOCK FB_System
VAR_INPUT
END_VAR
VAR_OUTPUT
END_VAR
VAR
	plcStart : PLC_Start;
	plcStop : PLC_Stop;
	plcReset : PLC_Reset;
END_VAR

{attribute 'TcRpcEnable'}
METHOD resetRuntime : BOOL
VAR_INPUT
END_VAR
plcReset(
	NETID:= , 
	PORT:= 851, 
	RESET:= TRUE, 
	TMOUT:= , 
	BUSY=> , 
	ERR=> , 
	ERRID=> );
	
plcReset(
	NETID:= , 
	PORT:= 851, 
	RESET:= FALSE, 
	TMOUT:= , 
	BUSY=> , 
	ERR=> , 
	ERRID=> );
END_METHOD

{attribute 'TcRpcEnable'}
METHOD startRuntime : BOOL
plcStart(
	NETID:= '', 
	PORT:= 851, 
	START:= TRUE, 
	TMOUT:= , 
	BUSY=> , 
	ERR=> , 
	ERRID=> );
	
plcStart(
	NETID:= '', 
	PORT:= 851, 
	START:= FALSE, 
	TMOUT:= , 
	BUSY=> , 
	ERR=> , 
	ERRID=> );
END_METHOD

{attribute 'TcRpcEnable'}
METHOD stopRuntime : BOOL
plcStop(
	NETID:= '', 
	PORT:= 851, 
	STOP:= TRUE, 
	TMOUT:= , 
	BUSY=> , 
	ERR=> , 
	ERRID=> );
	
plcStop(
	NETID:= '', 
	PORT:= 851, 
	STOP:= FALSE, 
	TMOUT:= , 
	BUSY=> , 
	ERR=> , 
	ERRID=> );
END_METHOD

END_FUNCTION_BLOCK

// ---- POUs/Materials/GetMaterialLength.TcPOU
FUNCTION GetMaterialLength : REAL
VAR_INPUT
	material : STRING;
END_VAR
VAR
	i : INT;
END_VAR

FOR i:=0 TO GVL.numMaterials BY 1 DO
	
	IF GVL.allMaterials[i].code = material THEN
		getMaterialLength := GVL.allMaterials[i].length;
		RETURN;
	END_IF
	
END_FOR
//otherwise, return 0
GetMaterialLength := 0;

END_FUNCTION

// ---- POUs/BundleToJson.TcPOU
PROGRAM BundleToJson
VAR
	fbJson : FB_JsonSaxWriter;
	fbJsonDataType : FB_JsonReadWriteDataType;
	jsonDoc : STRING(100000); //this wont even show up in online view as twincat cannot show strings this long
	arrDoc : ARRAY[0..100000] OF BYTE;
	
	newBundle : Bundle;
	getBundle : Bundle;
END_VAR

newBundle.id := 'abcdefghijkl';
newBundle.autoRE := TRUE;
newBundle.cardboard := MAIN.moduleA22.materialsArr;
newBundle.timeDone := MAIN.currentTime;

fbJson.ResetDocument();
fbJsonDataType.AddJsonValueFromSymbol(fbJson, 'Bundle', SIZEOF(newBundle), ADR(newBundle));
fbJson.CopyDocument(jsonDoc, SIZEOF(jsonDoc));

MEMCPY(
	ADR(arrDoc), 
	ADR(jsonDoc),
	MIN(
		SIZEOF(jsonDoc),
		SIZEOF(arrDoc))
	);
	
fbJsonDataType.SetSymbolFromJson(jsonDoc, 'Bundle', SIZEOF(getBundle), ADR(getBundle));

END_PROGRAM
